// TwinCAT 3 PLC project PLC1
// ProgramVersion: 3.1.4026.16
// CompilerDefines: VISU_USEPROPERTYINFO
// libraries:
//   SH_Light, * (StroemHansen)
//   Tc2_EnOcean, * (Beckhoff Automation GmbH)
//   Tc2_Standard, * (Beckhoff Automation GmbH)
//   Tc2_System, * (Beckhoff Automation GmbH)
//   Tc2_Utilities, * (Beckhoff Automation GmbH)
//   Tc3_DALI, * (Beckhoff Automation GmbH)
//   Tc3_System_DK, * (Beckhoff - DK)
//   VisuDialogs, * (System)
// project tree:
//   DUTs/DALI/ E_DALIExtendedFadeTime.TcTLEO (not stored), ST_DALI102Parameters.TcDUT (not stored), ST_DALI103Parameters.TcDUT (not stored), ST_DALIMemoryBank.TcDUT (not stored), ST_DALI_GrpAssignment.TcDUT (not stored), ST_GroupSort.TcDUT (not stored)
//   DUTs/EnOcean/ ST_ReadSAB05.TcDUT (not stored), ST_WriteSAB05.TcDUT (not stored)
//   / FastTask.TcTTO (not stored), GlobalTextList.TcGTLO (not stored), PlcTask.TcTTO (not stored), Visualization Manager.TcVMO (not stored)
//   GVLs/ GVL_AHDataModbus.TcGVL (not stored), GVL_EnOcean.TcGVL, GVL_Skalering.TcGVL (not stored)
//   POUs/01_System/01_System/GVLs/ GVL_EtherCAT.TcGVL (not stored)
//   POUs/01_System/01_System/ P_SystemDK.TcPOU (not stored)
//   POUs/AHModbusComm/ P_AHModbusComm.TcPOU
//   POUs/Alle_Rum/Gange/Gang_1_147/ P_Gang_1_147.TcPOU (not stored), Visualization_4_330_2_1.TcVIS (not stored) (excluded from build)
//   POUs/Alle_Rum/Gange/Gang_5_441/ P_Gang_5_441.TcPOU (not stored), Visualization_4_330_1_1_1_1_2_2.TcVIS (not stored) (excluded from build)
//   POUs/Alle_Rum/Gange/Gang_7_401/ P_Gang_7_401.TcPOU, Visualization_4_330_1.TcVIS (excluded from build)
//   POUs/Alle_Rum/Gange/Gang_6_210/ P_Gang_6_210.TcPOU, Visualization_4_308_1_2_1.TcVIS (not stored) (excluded from build)
//   POUs/Alle_Rum/Gange/Gang_4_413/ P_Gang_4_413.TcPOU, Visualization_4_330.TcVIS (not stored) (excluded from build)
//   POUs/Alle_Rum/Gange/Gang_1_148/ P_Gang_1_148.TcPOU (not stored), Visualization_4_330_2.TcVIS (not stored) (excluded from build)
//   POUs/Alle_Rum/Gange/Gang_4_434A/ P_Gang_4_434A.TcPOU, Visualization_4_330_1_1_1_1_2.TcVIS (not stored) (excluded from build)
//   POUs/Alle_Rum/Gange/Gang_5_441B/ P_Gang_5_441B.TcPOU, Visualization_5_338_1_2.TcVIS (not stored) (excluded from build)
//   POUs/Alle_Rum/Gange/Gang_Atrium/ P_Gang_Atrium.TcPOU (not stored), Visualization_5_338_2.TcVIS (not stored) (excluded from build)
//   POUs/Alle_Rum/Gange/Gang_5_238/ P_Gang_5_238.TcPOU (not stored), Visualization_5_338_1.TcVIS (not stored) (excluded from build)
//   POUs/Alle_Rum/Rum_Med_DALI_Pir/1_Rum_5_125_Og_5_127_Foldedoer/ P_Foldedoer_5_125.TcPOU (not stored), P_Rum_5_127.TcPOU (not stored), P_Rum_5_125.TcPOU (not stored), Visualization_5_352_1_1_1_1_1_1.TcVIS (not stored) (excluded from build)
//   POUs/Alle_Rum/Rum_Med_DALI_Pir/Rum_4_105/ P_Rum_4_105.TcPOU, Visualization_4_330_1_1_2_1.TcVIS (not stored) (excluded from build)
//   POUs/Alle_Rum/Rum_Med_DALI_Pir/Rum_4_109D/ P_Rum_4_109D.TcPOU, Visualization_4_330_1_1_1_1_2_1_1_1_2_1_1.TcVIS (not stored) (excluded from build)
//   POUs/Alle_Rum/Rum_Med_DALI_Pir/Rum_4_111A/ P_Rum_4_111A.TcPOU, Visualization_4_330_1_1_1_1_2_1_1_1_2_1_1_1.TcVIS (excluded from build)
//   POUs/Alle_Rum/Rum_Med_DALI_Pir/1Rum_5_448A/ P_Rum_5_448A.TcPOU (not stored), Visualization_4_330_1_1_1_1_2_1_1_1_3.TcVIS (not stored) (excluded from build)
//   POUs/Alle_Rum/Rum_Med_DALI_Pir/1Rum_5_444/ P_Rum_5_444.TcPOU (not stored), Visualization_4_308_1_2_1_1.TcVIS (excluded from build)
//   POUs/Alle_Rum/Rum_Med_DALI_Pir/Rum_4_107A/ P_Rum_4_107A.TcPOU, Visualization_4_330_1_1_1_1_2_1_1_1_1.TcVIS (excluded from build)
//   POUs/Alle_Rum/Rum_Med_DALI_Pir/1Rum_5_260B/ P_Rum_5_260B.TcPOU, Visualization_4_330_1_1_1_1_2_1_1.TcVIS (excluded from build)
//   POUs/Alle_Rum/Rum_Med_DALI_Pir/1Rum_1_428/ P_Rum_1_428.TcPOU, Visualization_5_338_1_1_1_1_2_1_1_1.TcVIS (excluded from build)
//   POUs/Alle_Rum/Rum_Med_DALI_Pir/Rum_4_109A/ P_Rum_4_109A.TcPOU, Visualization_4_330_1_1_1_1_2_1_1_1_2_1.TcVIS (not stored) (excluded from build)
//   POUs/Alle_Rum/Rum_Med_DALI_Pir/1Rum_4_426/ P_Rum_4_426.TcPOU (not stored), Visualization_4_330_1_1_1_1_2_1_1_1.TcVIS (not stored) (excluded from build)
//   POUs/Alle_Rum/Rum_Med_DALI_Pir/1Rum_5_456/ P_Rum_5_456.TcPOU, Visualization_4_330_1_1_1_1_2_1_1_1_3_1_1_1_1_1.TcVIS (not stored) (excluded from build)
//   POUs/Alle_Rum/Rum_Med_DALI_Pir/1Rum_5_450/ P_Rum_5_450.TcPOU (not stored), Visualization_4_330_1_1_1_1_2_1_1_1_3_1.TcVIS (not stored) (excluded from build)
//   POUs/Alle_Rum/Rum_Med_DALI_Pir/1Rum_5_448B/ P_Rum_5_448B.TcPOU, Visualization_4_330_1_1_1_1_2_1.TcVIS (not stored) (excluded from build)
//   POUs/Alle_Rum/Rum_Med_DALI_Pir/1Rum_5_452/ P_Rum_5_452.TcPOU (not stored), Visualization_4_330_1_1_1_1_2_1_1_1_3_1_1.TcVIS (not stored) (excluded from build)
//   POUs/Alle_Rum/Rum_Med_DALI_Pir/1Rum_5_454/ P_Rum_5_454.TcPOU (not stored), Visualization_4_330_1_1_1_1_2_1_1_1_3_1_1_1.TcVIS (not stored) (excluded from build)
//   POUs/Alle_Rum/Rum_Med_DALI_Pir/1Rum_5_450B/ P_Rum_5_450B.TcPOU (not stored), Visualization_4_330_1_1_1_1_2_1_1_1_3_1_1_1_1.TcVIS (not stored) (excluded from build)
//   POUs/Alle_Rum/Rum_Med_DALI_Pir/1Rum_5_411C/ P_Rum_5_411C.TcPOU (not stored), Visualization_4_330_1_1_1_1_2_1_1_1_3_1_1_1_1_1_1.TcVIS (excluded from build)
//   POUs/Alle_Rum/Rum_Med_DALI_Pir/1Rum_6_205/ P_Rum_6_205.TcPOU (not stored), Visualization_5_338_1_1_2_1_1_1_1_1_1_1_1_1_1_1_1_2_2_1_1.TcVIS (not stored) (excluded from build)
//   POUs/Alle_Rum/Rum_Med_DALI_Pir/1Rum_5_441A/ P_Rum_5_441A.TcPOU (not stored), Visualization_5_338_1_1_2_1_1_1_1_1_1_1_1_1_1_1_1_2_2_2.TcVIS (not stored) (excluded from build)
//   POUs/Alle_Rum/Rum_Med_DALI_Pir/1Rum_5_263/ P_Rum_5_263.TcPOU (not stored), Visualization_5_338_1_1_2_1_1_1_1_1_1_1_1_1_1_1_1_2_2_1.TcVIS (excluded from build)
//   POUs/Alle_Rum/Rum_Med_DALI_Pir/1Rum_3_155/ P_Rum_3_155.TcPOU (not stored), Visualization_5_352_1_1_1_1_1_2_1.TcVIS (not stored) (excluded from build)
//   POUs/Alle_Rum/Rum_Med_DALI_Pir/1Rum_6_214B/ P_Rum_6_214B.TcPOU (not stored), Visualization_4_330_1_1_1_1_2_1_1_1_2.TcVIS (excluded from build)
//   POUs/Alle_Rum/Trapper/ P_Trappe_T4.TcPOU
//   POUs/DALI/DALI_Setup/ DALI_Commissioning.TcPOU (not stored)
//   POUs/DALI/DALI_Setup/FBs/ FB_Part102Addressing.TcPOU (not stored), FB_Part102Commands.TcPOU (not stored), FB_Part102Groups.TcPOU (not stored), FB_Part102MemoryPages.TcPOU (not stored), FB_Part102Parameters.TcPOU (not stored), FB_Part102Scenes.TcPOU (not stored), FB_Part102SetFading.TcPOU (not stored), FB_Part103Addressing.TcPOU (not stored), FB_Part103MemoryPages.TcPOU (not stored), FB_Part103Identify.TcPOU (not stored), FB_Part103Parameters.TcPOU (not stored), FB_Part202Emergency.TcPOU (not stored), FB_Part205Incandescent.TcPOU (not stored), FB_Part207LED.TcPOU (not stored), FB_Part208Switching.TcPOU (not stored), FB_Part300GenericDevice.TcPOU (not stored), FB_Part301PushButton.TcPOU (not stored), FB_Part302AbsoluteInputDevice.TcPOU (not stored), FB_Part303OccupancySensor.TcPOU (not stored), FB_Part304LightSensor.TcPOU (not stored), GearType.TcPOU (not stored)
//   POUs/DALI/DALI_Setup/GVLs/ GVL_Internal.TcGVL (not stored)
//   POUs/DALI/DALI_Setup/VISUs/TextLists/ CommandOnTerminalEvent.TcTLO (not stored), DimmingCurve.TcTLO, EventPriority.TcTLO (not stored), EventScheme.TcTLO (not stored), ExtendedFadeTime.TcTLO (not stored), FadeRate.TcTLO (not stored), FadeTime.TcTLO (not stored), FastFadeTime.TcTLO (not stored), TextList_Dialogs.TcTLO (not stored)
//   POUs/DALI/DALI_Setup/VISUs/ Visu_DALICommissioning.TcVIS (not stored)
//   POUs/DALI/DALI_Setup/VISUs/Visu_DALICommissioning/ Visu_KL6821Configuration.TcVIS (not stored) (excluded from build), Visu_Part102Addressing.TcVIS (not stored), Visu_Part102Commands.TcVIS (not stored), Visu_Part102Groups.TcVIS (not stored), Visu_Part102MemoryBank.TcVIS (not stored), Visu_Part102Parameters.TcVIS (not stored), Visu_Part102Scenes.TcVIS (not stored), Visu_Part102SetFading.TcVIS (not stored), Visu_Part103Addressing.TcVIS (not stored), Visu_Part103Identify.TcVIS (not stored), Visu_Part103MemoryBank.TcVIS (not stored), Visu_Part103Parameters.TcVIS (not stored), Visu_Part202.TcVIS (not stored), Visu_Part202Commands.TcVIS (not stored), Visu_Part202Parameters.TcVIS (not stored), Visu_Part202Status.TcVIS (not stored), Visu_Part205.TcVIS (not stored), Visu_Part205Parameters.TcVIS (not stored), Visu_Part205Status.TcVIS (not stored), Visu_Part207.TcVIS (not stored), Visu_Part207Parameters.TcVIS (not stored), Visu_Part207Status.TcVIS (not stored), Visu_Part208Switching.TcVIS (not stored), Visu_Part300GenericDevice.TcVIS (not stored), Visu_Part301PushButton.TcVIS (not stored), Visu_Part302AbsoluteInputDevice.TcVIS (not stored), Visu_Part303OccupancySensor.TcVIS (not stored), Visu_Part304LightSensor.TcVIS (not stored), Visu_Welcome.TcVIS (not stored)
//   POUs/DALI/PRGs/Background/ P_DALI_Background.TcPOU (not stored)
//   POUs/DALI/PRGs/Diag/ P_DALI_DIAG.TcPOU (not stored)
//   POUs/DALI/PRGs/EnergyData/ P_DALI_Energy_Firmware_Test.TcPOU (not stored) (excluded from build), P_DALI_Energy_Line.TcPOU (not stored)
//   POUs/EnOcean/ P_EnOcean.TcPOU
//   POUs/ MAIN.TcPOU
// real-time tasks:
//   TASK PlcTask: cycle T#40ms, priority 21, ADS port 350
//   TASK FastTask: cycle T#4ms, priority 20, ADS port 351
// I/O:
//   DEVICE Device 1 (Beckhoff CCAT)
//   DEVICE Device 3 (CX-BK)
//     Box 1 (CX-BK)
// variable links:
//   PLC1/PLC1 Instance <-> Device 3 (CX-BK)/Box 1 (CX-BK)
//     FastTask Inputs/P_DALI_Background.arrKL6821InData[1] @bit 16 <-> Term 5 (KL6821)/Channel 1/Data In 0
//     FastTask Inputs/P_DALI_Background.arrKL6821InData[1] @bit 24 <-> Term 5 (KL6821)/Channel 1/Data In 1
//     FastTask Inputs/P_DALI_Background.arrKL6821InData[1] @bit 32 <-> Term 5 (KL6821)/Channel 1/Data In 2
//     FastTask Inputs/P_DALI_Background.arrKL6821InData[1] @bit 40 <-> Term 5 (KL6821)/Channel 1/Data In 3
//     FastTask Inputs/P_DALI_Background.arrKL6821InData[2] @bit 16 <-> Term 6 (KL6821)/Channel 1/Data In 0
//     FastTask Inputs/P_DALI_Background.arrKL6821InData[2] @bit 24 <-> Term 6 (KL6821)/Channel 1/Data In 1
//     FastTask Inputs/P_DALI_Background.arrKL6821InData[2] @bit 32 <-> Term 6 (KL6821)/Channel 1/Data In 2
//     FastTask Inputs/P_DALI_Background.arrKL6821InData[2] @bit 40 <-> Term 6 (KL6821)/Channel 1/Data In 3
//     FastTask Inputs/P_DALI_Background.arrKL6821InData[1] <-> Term 5 (KL6821)/Channel 1/State
//     FastTask Inputs/P_DALI_Background.arrKL6821InData[2] <-> Term 6 (KL6821)/Channel 1/State
//     FastTask Inputs/P_EnOcean.stKL6581_in @bit 8 <-> Term 3 (KL6581)/Channel 1/Input CNODE
//     FastTask Inputs/P_EnOcean.stKL6581_in @bit {24..48 step 8} <-> Term 3 (KL6581)/Channel 1/Input DB{0..3}  (4 links)
//     FastTask Inputs/P_EnOcean.stKL6581_in @bit {56..80 step 8} <-> Term 3 (KL6581)/Channel 1/Input ID{0..3}  (4 links)
//     FastTask Inputs/P_EnOcean.stKL6581_in @bit 16 <-> Term 3 (KL6581)/Channel 1/Input ORG
//     FastTask Inputs/P_EnOcean.stKL6581_in @bit 88 <-> Term 3 (KL6581)/Channel 1/Input STATUS
//     FastTask Inputs/P_EnOcean.stKL6581_in <-> Term 3 (KL6581)/Channel 1/Status
//     FastTask Outputs/P_DALI_Background.arrKL6821OutData[1] <-> Term 5 (KL6821)/Channel 1/Ctrl
//     FastTask Outputs/P_DALI_Background.arrKL6821OutData[2] <-> Term 6 (KL6821)/Channel 1/Ctrl
//     FastTask Outputs/P_DALI_Background.arrKL6821OutData[1] @bit 16 <-> Term 5 (KL6821)/Channel 1/Data Out 0
//     FastTask Outputs/P_DALI_Background.arrKL6821OutData[1] @bit 24 <-> Term 5 (KL6821)/Channel 1/Data Out 1
//     FastTask Outputs/P_DALI_Background.arrKL6821OutData[1] @bit 32 <-> Term 5 (KL6821)/Channel 1/Data Out 2
//     FastTask Outputs/P_DALI_Background.arrKL6821OutData[1] @bit 40 <-> Term 5 (KL6821)/Channel 1/Data Out 3
//     FastTask Outputs/P_DALI_Background.arrKL6821OutData[2] @bit 16 <-> Term 6 (KL6821)/Channel 1/Data Out 0
//     FastTask Outputs/P_DALI_Background.arrKL6821OutData[2] @bit 24 <-> Term 6 (KL6821)/Channel 1/Data Out 1
//     FastTask Outputs/P_DALI_Background.arrKL6821OutData[2] @bit 32 <-> Term 6 (KL6821)/Channel 1/Data Out 2
//     FastTask Outputs/P_DALI_Background.arrKL6821OutData[2] @bit 40 <-> Term 6 (KL6821)/Channel 1/Data Out 3
//     FastTask Outputs/P_EnOcean.stKL6581_out <-> Term 3 (KL6581)/Channel 1/Control
//     FastTask Outputs/P_EnOcean.stKL6581_out @bit 8 <-> Term 3 (KL6581)/Channel 1/Output CNODE
//     FastTask Outputs/P_EnOcean.stKL6581_out @bit {24..48 step 8} <-> Term 3 (KL6581)/Channel 1/Output DB{0..3}  (4 links)
//     FastTask Outputs/P_EnOcean.stKL6581_out @bit {56..80 step 8} <-> Term 3 (KL6581)/Channel 1/Output ID{0..3}  (4 links)
//     FastTask Outputs/P_EnOcean.stKL6581_out @bit 16 <-> Term 3 (KL6581)/Channel 1/Output ORG
//     FastTask Outputs/P_EnOcean.stKL6581_out @bit 88 <-> Term 3 (KL6581)/Channel 1/Output STATUS
//     PlcTask Inputs/MAIN.nCX8200_State <-> Inputs/State
//     PlcTask Inputs/P_Trappe_T4.bDigitalPir <-> Term 4 (KL1408)/Channel 1/Input
//     PlcTask Outputs/P_Trappe_T4.bTrappelysNC <-> Term 2 (KL2012)/Channel 1/Output

// ---- GVLs/GVL_EnOcean.TcGVL
{attribute 'qualified_only'}
VAR_GLOBAL
	
//Atrium
	strEnOceanSwitch_AtriumNiveau_PladeB				: Tc2_EnOcean.STR_EnOceanSwitch;
	strEnOceanSwitch_AtriumNiveau_Service				: Tc2_EnOcean.STR_EnOceanSwitch;


//Gange
//	strEnOceanSwitch_Gang_3_364				: Tc2_EnOcean.STR_EnOceanSwitch;

	//
 
     strEnOceanSwitch_Rum_4_105                      	: Tc2_EnOcean.STR_EnOceanSwitch;


END_VAR

// ---- POUs/AHModbusComm/P_AHModbusComm.TcPOU
PROGRAM P_AHModbusComm
VAR
	arrfbReadAHPirData	: ARRAY[1..GVL_AHDataModbus.byNumberOfAH_Neighbors] OF SH_Light.FB_ReadAHPirData;
	arrReadAHPirData		: ARRAY[1..GVL_AHDataModbus.byNumberOfAH_Neighbors] OF BOOL;
	
	arrfbTriggerPulses			: ARRAY[1..GVL_AHDataModbus.byNumberOfAH_Neighbors] OF SH_Light.FB_ClockPulse;
	arrGeneratePulses			: ARRAY[1..GVL_AHDataModbus.byNumberOfAH_Neighbors] OF BOOL := [GVL_AHDataModbus.byNumberOfAH_Neighbors(TRUE)];
	tTimeInterval					: TIME := T#1S;
	tPulseTime					: TIME := T#1S;
	
	byLineId						: BYTE;
	byAHId						: BYTE;
		fbWritePirDelayTime		: R_TRIG;
	bRunOverrideOnce		: BOOL := FALSE;
	bEnableDelayTimeOverride : BOOL := FALSE;
	uiPirOffDelayTimeAllRooms : UINT := 30;
	
END_VAR

VAR CONSTANT
	arrnMBAddr					: ARRAY[1..GVL_AHDataModbus.byNumberOfAH_Neighbors] OF WORD := [GVL_AHDataModbus.byNumberOfAH_Neighbors(12588)]; //modbus-adresser (%MB600=>12588 default)
	arrstNeighborIPAddr		: ARRAY[1..GVL_AHDataModbus.byNumberOfAH_Neighbors] OF SH_Light.ST_NeighborIP := [
																						(sPLCName := 'AH1-1', sIP := '172.24.195.161', IsNeighbor := FALSE), 
																				     	(sPLCName := 'AH1-2', sIP := '172.24.195.162', IsNeighbor := FALSE), 
																						(sPLCName := 'AH1-3', sIP := '172.24.195.163', IsNeighbor := FALSE),
																						(sPLCName := 'AH2-1', sIP := '172.24.195.164', IsNeighbor := FALSE),
																					    (sPLCName := 'AH2-2', sIP := '172.24.195.165', IsNeighbor := FALSE),
																						(sPLCName := 'AH2-3', sIP := '172.24.195.166', IsNeighbor := FALSE),
																				        (sPLCName := 'AH2-4', sIP := '172.24.195.167', IsNeighbor := FALSE),
																						(sPLCName := 'AH2-5', sIP := '172.24.195.168', IsNeighbor := FALSE),
																						(sPLCName := 'AH3-2', sIP := '172.24.195.169', IsNeighbor := FALSE),
																						(sPLCName := 'AH3-3', sIP := '172.24.195.170', IsNeighbor := FALSE),
																			         	(sPLCName := 'AH3-4', sIP := '172.24.195.171', IsNeighbor := FALSE),
																						(sPLCName := 'AH3-5', sIP := '172.24.195.172', IsNeighbor := FALSE),
																						(sPLCName := 'AH4-1', sIP := '172.24.195.173', IsNeighbor := FALSE),
																						(sPLCName := 'AH4-2', sIP := '172.24.195.174', IsNeighbor := FALSE),
																						(sPLCName := 'AH4-3', sIP := '172.24.195.175', IsNeighbor := FALSE),
																			            (sPLCName := 'AH4-4', sIP := '172.24.195.176', IsNeighbor := FALSE),
																						(sPLCName := 'AH4-5', sIP := '172.24.195.177', IsNeighbor := FALSE),
																						(sPLCName := 'AH5-1', sIP := '172.24.195.178', IsNeighbor := FALSE),
																					    (sPLCName := 'AH5-2', sIP := '172.24.195.179', IsNeighbor := FALSE), 
																						(sPLCName := 'AH5-3', sIP := '172.24.195.180', IsNeighbor := FALSE),
																						(sPLCName := 'AH5-4', sIP := '172.24.195.181', IsNeighbor := FALSE),
																						(sPLCName := 'AH5-5', sIP := '172.24.195.182', IsNeighbor := FALSE),
																						(sPLCName := 'AH6-1', sIP := '172.24.195.183', IsNeighbor := FALSE),
																				        (sPLCName := 'AH6-2', sIP := '172.24.195.184', IsNeighbor := FALSE),//Local must be false
																				(sPLCName := 'AH6-3', sIP := '172.24.195.185', IsNeighbor := FALSE)];
																					//	(sPLCName := 'AH3-1', sIP := '172.24.195.186', IsNeighbor := TRUE) //when ready
END_VAR

A_AHNeighborRoomsPirIn();
A_AHNeighborRoomsPirOut();
A_DALILineShrtAddrErr();
A_DelayTimeAllRooms();

ACTION A_AHNeighborRoomsPirIn:
FOR byAHId := 1 TO GVL_AHDataModbus.byNumberOfAH_Neighbors DO
	IF arrstNeighborIPAddr[byAHId].IsNeighbor THEN
		//Generate Pulses
		arrfbTriggerPulses[byAHId](bGenerateClockPulses:= arrGeneratePulses[byAHId], tTimeInterval:= tTimeInterval, tPulseTime:= tPulseTime);
		arrReadAHPirData[byAHId]:= arrfbTriggerPulses[byAHId].bPulse;
		//Read data
		arrfbReadAHPirData[byAHId](	bReadAHPirData				:=	arrReadAHPirData[byAHId],
														sIPAddr							:=	arrstNeighborIPAddr[byAHId].sIP,
														nMBAddr							:=	arrnMBAddr[byAHId],
														nMBDataBuffer				:=	GVL_AHDataModbus.arrAH_NeighborRoomsPir_In[byAHId],
														arrAH_NeighborRoomsPir	=>GVL_AHDataModbus.arrAH_NeighborRoomsPir[byAHId]);
	END_IF
END_FOR
END_ACTION

ACTION A_AHNeighborRoomsPirOut:
//GVL_AHDataModbus.nAH_NeighborRoomsPir_Out.0 := P_Gang_4_413.bPirActive_MB;
//GVL_AHDataModbus.nAH_NeighborRoomsPir_Out.1 := P_Gang_7_401.bPirActive_MB;
//GVL_AHDataModbus.nAH_NeighborRoomsPir_Out.2 := P_Gang_5_441.bPirActive_MB;
//GVL_AHDataModbus.nAH_NeighborRoomsPir_Out.3 := P_Rum_4_424.bPirActive_MB;
//GVL_AHDataModbus.nAH_NeighborRoomsPir_Out.4 := P_Rum_4_426.bPirActive_MB;
//GVL_AHDataModbus.nAH_NeighborRoomsPir_Out.5 := 
//GVL_AHDataModbus.nAH_NeighborRoomsPir_Out.6 :=
//GVL_AHDataModbus.nAH_NeighborRoomsPir_Out.7 := 
//GVL_AHDataModbus.nAH_NeighborRoomsPir_Out.8 :=
//GVL_AHDataModbus.nAH_NeighborRoomsPir_Out.9 := 
//GVL_AHDataModbus.nAH_NeighborRoomsPir_Out.10 :=
//GVL_AHDataModbus.nAH_NeighborRoomsPir_Out.11 := 
//GVL_AHDataModbus.nAH_NeighborRoomsPir_Out.12 := 
//GVL_AHDataModbus.nAH_NeighborRoomsPir_Out.13 := 
//GVL_AHDataModbus.nAH_NeighborRoomsPir_Out.14 := 
//GVL_AHDataModbus.nAH_NeighborRoomsPir_Out.15 :=
END_ACTION

ACTION A_DALILineShrtAddrErr:
FOR  byLineId := 1 TO SH_Light.DALI_Param.MAX_DALIV2_LINES DO
	GVL_AHDataModbus.arrDALILineShrtAddrErr[byLineId] :=  TO_UINT(SH_Light.GVL_DALI_LatestError.arrLineShrtAddr[byLineId]);
END_FOR
END_ACTION

ACTION A_DelayTimeAllRooms:

fbWritePirDelayTime(CLK := GVL_AHDataModbus.uiPirOffDelayTimeAllRooms_MB<>uiPirOffDelayTimeAllRooms);

IF fbWritePirDelayTime.Q THEN
	bRunOverrideOnce := TRUE;
	bEnableDelayTimeOverride := TRUE;
	
//Indsæt kode
P_Rum_4_105.fbWritePirDelayTIme(bEnableOverride := bEnableDelayTimeOverride, nOverRideValue := GVL_AHDataModbus.uiPirOffDelayTimeAllRooms_MB, nValIn1 := GVL_AHDataModbus.uiPirOffDelayTimeAllRooms_MB, nValIn2 := uiPirOffDelayTimeAllRooms);
P_Rum_4_107A.fbWritePirDelayTIme(bEnableOverride := bEnableDelayTimeOverride, nOverRideValue := GVL_AHDataModbus.uiPirOffDelayTimeAllRooms_MB, nValIn1 := GVL_AHDataModbus.uiPirOffDelayTimeAllRooms_MB, nValIn2 := uiPirOffDelayTimeAllRooms);
P_Rum_4_109A.fbWritePirDelayTIme(bEnableOverride := bEnableDelayTimeOverride, nOverRideValue := GVL_AHDataModbus.uiPirOffDelayTimeAllRooms_MB, nValIn1 := GVL_AHDataModbus.uiPirOffDelayTimeAllRooms_MB, nValIn2 := uiPirOffDelayTimeAllRooms);
P_Rum_4_109D.fbWritePirDelayTIme(bEnableOverride := bEnableDelayTimeOverride, nOverRideValue := GVL_AHDataModbus.uiPirOffDelayTimeAllRooms_MB, nValIn1 := GVL_AHDataModbus.uiPirOffDelayTimeAllRooms_MB, nValIn2 := uiPirOffDelayTimeAllRooms);
P_Rum_4_111A.fbWritePirDelayTIme(bEnableOverride := bEnableDelayTimeOverride, nOverRideValue := GVL_AHDataModbus.uiPirOffDelayTimeAllRooms_MB, nValIn1 := GVL_AHDataModbus.uiPirOffDelayTimeAllRooms_MB, nValIn2 := uiPirOffDelayTimeAllRooms);



ELSE
	IF bRunOverrideOnce THEN
		bEnableDelayTimeOverride := FALSE;
		
		//Indsæt kode
P_Rum_4_105.fbWritePirDelayTIme(bEnableOverride := bEnableDelayTimeOverride, nOverRideValue := GVL_AHDataModbus.uiPirOffDelayTimeAllRooms_MB, nValIn1 := GVL_AHDataModbus.uiPirOffDelayTimeAllRooms_MB, nValIn2 := uiPirOffDelayTimeAllRooms);
P_Rum_4_107A.fbWritePirDelayTIme(bEnableOverride := bEnableDelayTimeOverride, nOverRideValue := GVL_AHDataModbus.uiPirOffDelayTimeAllRooms_MB, nValIn1 := GVL_AHDataModbus.uiPirOffDelayTimeAllRooms_MB, nValIn2 := uiPirOffDelayTimeAllRooms);
P_Rum_4_109A.fbWritePirDelayTIme(bEnableOverride := bEnableDelayTimeOverride, nOverRideValue := GVL_AHDataModbus.uiPirOffDelayTimeAllRooms_MB, nValIn1 := GVL_AHDataModbus.uiPirOffDelayTimeAllRooms_MB, nValIn2 := uiPirOffDelayTimeAllRooms);
P_Rum_4_109D.fbWritePirDelayTIme(bEnableOverride := bEnableDelayTimeOverride, nOverRideValue := GVL_AHDataModbus.uiPirOffDelayTimeAllRooms_MB, nValIn1 := GVL_AHDataModbus.uiPirOffDelayTimeAllRooms_MB, nValIn2 := uiPirOffDelayTimeAllRooms);
P_Rum_4_111A.fbWritePirDelayTIme(bEnableOverride := bEnableDelayTimeOverride, nOverRideValue := GVL_AHDataModbus.uiPirOffDelayTimeAllRooms_MB, nValIn1 := GVL_AHDataModbus.uiPirOffDelayTimeAllRooms_MB, nValIn2 := uiPirOffDelayTimeAllRooms);

		bRunOverrideOnce := FALSE;
		
		
	END_IF
END_IF
END_ACTION

END_PROGRAM

// ---- POUs/Alle_Rum/Rum_Med_DALI_Pir/Rum_4_105/P_Rum_4_105.TcPOU
PROGRAM P_Rum_4_105
VAR

	fbLys		: FB_Light_Type_A;
	

	stDaliSetup	: SH_Light.ST_DALI_RoomSetup := (	
														byShrtAdr_Prim := 1, 
														byGrpAdr_Prim := 1, 
														eMod_Prim := E_DALIAddressType.Group, 
														//byShrtAdr_Sec := 1, 
														//byGrpAdr_Sec := 1, 
														//eMod_Sec := E_DALIAddressType.Short, 
														//byShrtAdr_Supl := 1, 
														DALI_LINE_NUM_PRIM := DALI_LINE_NUM_LIGHT,
														DALI_LINE_NUM_SEC := 0, //0 = ingen zonestyring/vinduerække
														DALI_LINE_NUM_SUPL := DALI_LINE_NUM_PENDANTS);
														
	stLiveData					: SH_Light.ST_LiveData;
	bRunTuning					: BOOL;
	
	bTopButtonZone1				: BOOL;
	bTopButtonZone1_Visu		: BOOL;
	bBottomButtonZone1			: BOOL;
	bBottomButtonZone1_Visu	: BOOL;
	bButtonZone2				: BOOL;
	fLuxOn							: REAL;
	fLuxDim						: REAL;
	tPIRDim						: TIME;
	tPIROff						: TIME;
	fOffsetSec					: REAL := 20;
	bOccupiedRoom			: BOOL;;


// Sensor Settings
	//fbSensor						: SH_Light.FB_NIKO_P46xx_1Pcs;
	fbSensor						: SH_Light.FB_NIKO_P46xx_3Pcs;
	//bySensorAddr				: BYTE := 8;
	arrSensorAddr				: ARRAY[1..3] OF BYTE := [1,2,3];
	bInitialize						: BOOL := TRUE;
	stDaliSensorSetup			: ST_DALI_NIKOP46SetupData := (
																nSensitivityPIRSegmentA := arrSensitivityOccupancy[1],
																nSensitivityPIRSegmentB := arrSensitivityOccupancy[2],
																nSensitivityPIRSegmentC := arrSensitivityOccupancy[3]);
	//bInitErr							: BOOL;
	//bInitDone						: BOOL;
	arrInitErr						: ARRAY [1..3] OF BOOL;
	arrInitDone					: ARRAY [1..3] OF BOOL;
	arrSensorScales				: ARRAY [1..10] OF SH_Light.ST_DALI_SensorScaleMode := [
																						(fMeassureMaxSensor := rMeassure_Zone5, fReadMaxSensor := rRead_Zone5),	
																						(fMeassureMaxSensor := rMeassure_Zone5, fReadMaxSensor := rRead_Zone5),	
																						(fMeassureMaxSensor := rMeassure_Zone5, fReadMaxSensor := rRead_Zone5),																																										
																						7(())];
	bCancelHoldTimerOccupancy	: BOOL;
(*	eEventPriorityOccupancy		: E_DALIEventPriority := E_DALIEVENTPRIORITY.Middle;
	nHoldTimerOccupancy			: WORD := 5; // Value in s. 	
	nReportTimerOccupancy		: BYTE := 120; // Value in s, Preset manufacturer value
	nDeadtimeTimerOccupancy		: WORD := 100; // Value in ms, Predefined Value of DALI Standard
	bCancelHoldTimerOccupancy	: BOOL;
	nSensitivityOccupancy		: BYTE:= 3; //setting Sensivity (0..4) 0 (Off), 1 (Min), 2(Low), 3(High) and 4 (Max)

	bEnableLuxEvent				: BOOL;
	eEventPriorityBrightness	: E_DALIEventPriority := E_DALIEVENTPRIORITY.Middle;
	nDeadtimeTimerBrightness	: WORD := 1500; // Value in ms, Predefined Value of DALI Standard
	nHysteresisBrightness		: BYTE := 2; // Value in %
	nHysteresisMinBrightness	: BYTE := 10; // Absolute Value, depending on the manufacturer specific resolution
	nReportTimerBrightness		: BYTE := 120; // Value in s, Preset manufacturer value
*)

	//stDaliSetup: SH_Light.ST_DALI_RoomSetup
	//stRoomDataModbus			: SH_Light.ST_RoomDataModbus := ( bPirActive := bPirActive
	

	//ModbusComm setup
	
	fbWriteSPLuxLevel			: SH_Light.FB_TwoVal_SelectOne_RTrigChange;
	fbWritePirDelayTIme		: SH_Light.FB_TwoVal_SelectOne_RTrigChange;
	stRoomDataPLC				: SH_Light.ST_RoomDataPLC	:=	(
																	uiPirOffDelayTime	:= 30,
																	uiSpLuxLevel			:= 500,
																	uiPirDimDelayTime	:= 15,
																	uiSpDimLuxLevel		:= 200);
																	
	fbBallastOnHours				: SH_Light.FB_CountOnHours;
	bEnableHourCount			: BOOL := TRUE;
	
	//Non-persistent modbus data
	bPirActive_MB					AT %MX0.0	: BOOL;				//bPirLys i gammel kode
	uiActLuxLevel_MB			AT %MB4	: UINT;				//intHMIAktueltLux i gammel kode
	uiActLightLevelPct_MB	AT %MB10		: UINT;				//intDALI_Gruppe1_Lysniveau i gammel kode
	
	//For Conversion
	uiPirOffMinutes						: UINT;
	udTimeScaling						: UDINT := 60000;
	uiLuxOn								: UINT;
	
	//max values checks
	uiMaxLuxLevel						: UINT := 1023;
	uiMaxPirOffMinutes				: UINT := 180;

	
END_VAR

VAR CONSTANT
    Sensor_DALI_LINE_NUM				: BYTE := 1;
	DALI_LINE_NUM_LIGHT				: BYTE := 1;
    DALI_LINE_NUM_PENDANTS	: BYTE := 0; //0=ingen pendler
	arrSensitivityOccupancy						: ARRAY[1..3] OF BYTE := [4,4,4]; //setting Sensivity (0..4) 0 (Off), 1 (Min), 2(Low), 3(High) and 4 (Max)
END_VAR
VAR PERSISTENT
	stPirSensorData: SH_Light.ST_DALI_Sensor;
	stTuneData: SH_Light.ST_TuneData_EX;

	uiPirOffDelayTime_MB		AT %MB2		: UINT;				//ntHMI_Pir_SetValue i gammel kode
	uiSPLuxLevel_MB			AT %MB6	: UINT;				//intHMI_Lux_SetValue i gammel kode
	uiBallastOnHours_MB		AT %MB14		: UINT;				//dintHMILysbraendtimer1 i gammel kode
	byOnHoursOverflowCount							: BYTE;   
END_VAR

A_Buttons();
A_LightCtrl();
A_Sensor();
A_ModbusComm();

ACTION A_Buttons:
bTopButtonZone1		:= GVL_EnOcean.strEnOceanSwitch_Rum_4_105.bT1_ON OR  bTopButtonZone1_Visu;
bBottomButtonZone1	:= GVL_EnOcean.strEnOceanSwitch_Rum_4_105.bT1_OFF OR  bBottomButtonZone1_Visu;
END_ACTION

ACTION A_LightCtrl:
fbLys(
	nZoneID:= 1, 
	bButtonZone1:= bTopButtonZone1,
	bBottomButtonZone1 := bBottomButtonZone1, 
	//bButtonZone2:= bButtonZone2,
	fLuxOn:= fLuxOn, 
	fLuxDim:= fLuxDim, 
	tPIRDim:= tPIRDim, 
	tPIROff:= tPIROff, 
	fOffsetSec:= fOffsetSec, 
	bReInit:= , 
	stDaliSetup:= stDaliSetup, 
	ipCommunication_Prim:= P_DALI_Background.arrfbKL6821Communication[DALI_LINE_NUM_LIGHT], 
	//ipCommunication_Sec:= P_DALI_Background.arrfbKL6821Communication[DALI_LINE_NUM_LIGHT], 
	//ipCommunication_Supl:= P_DALI_Background.arrfbKL6821Communication[DALI_LINE_NUM_PENDANTS], 
	fMinOutputPowerLevelRoom:= 15, 
	fMaxOutputPowerLevelRoom:= 100, 
	nCycleTimeInMS:= SH_Light.DALI_Param.nPlcTaskCycleTimeInMS*nDimCmdCycleTimeFactor , 
	bRunTuning:= bRunTuning, 
	bOccupiedRoom=> bOccupiedRoom, 
	bError_Prim=> , 
	nError_Prim=> , 
	stTuneData:=stTuneData , 
	stPirSensorData:= stPirSensorData, 
	stLiveData:= stLiveData);
END_ACTION

ACTION A_ModbusComm:
//Manage data for modbus communication

//Manage data for read-only in PLC
stRoomDataPLC.bPirActive			:= stPirSensorData.bPrc;
stRoomDataPLC.uiActLuxLevel			:= TO_UINT(TRUNC(stPirSensorData.fBrightness));
stRoomDataPLC.uiActLightLevelPct	:= TO_UINT(TRUNC(fbLys.fbBallast.fActlLgtLvl_Prim));
		//stRoomDataPLC.uiActLightLevelPct	:= TO_UINT(TRUNC(fbLys.fbBallast.fActlLgtLvl_Prim)); //if only one group light control
stRoomDataPLC.uiBallastOnHours		:= uiBallastOnHours_MB; //The calculation for BallastOnHours is stored directly to the MB register below


//Assign data for read-only to MB registers
bPirActive_MB			:= stRoomDataPLC.bPirActive;
uiActLuxLevel_MB		:= stRoomDataPLC.uiActLuxLevel;
uiActLightLevelPct_MB	:= stRoomDataPLC.uiActLightLevelPct;

	//calculate BallastOnHours
	fbBallastOnHours(
		bEnableHourCount	:= bEnableHourCount,
		bPauseCount			:= fbLys.fbLightCtrl.bOffZone1,
		uiOnHours			:= uiBallastOnHours_MB,			//OnHours is updated here
		byOverflowCount		:= byOnHoursOverflowCount);


//Manage data for read/write for both PLC and MB registers
fbWriteSPLuxLevel(	nMaxValOut	:= uiMaxLuxLevel,
					nValIn1		:= uiSPLuxLevel_MB,		//nValIn1 takes priotity in case of download or restart
					nValIn2		:= stRoomDataPLC.uiSpLuxLevel,
					nValOut		=> uiLuxOn
				);


fbWritePirDelayTIme(	nMaxValOut	:= uiMaxPirOffMinutes,
						nValIn1		:= uiPirOffDelayTime_MB,		//nValIn1 takes priotity in case of download or restart
						nValIn2		:= stRoomDataPLC.uiPirOffDelayTime,
						nValOut		=> uiPirOffMinutes
					);
					

//Convert read/write modbus data to appropriate datatypes in PLC
fLuxOn	:= TO_REAL(uiLuxOn);			
tPIROff	:= TO_TIME(uiPirOffMinutes*udTimeScaling); //Time conversion defaults to ms

fLuxDim	:= TO_REAL(stRoomDataPLC.uiSpDimLuxLevel);			
tPIRDim	:= TO_TIME(stRoomDataPLC.uiPirDimDelayTime*udTimeScaling); //Time conversion defaults to ms
END_ACTION

ACTION A_Sensor:

fbSensor.ipCommunication := P_DALI_Background.arrfbKL6821Communication[Sensor_DALI_LINE_NUM];

//only 1 sensor
(*fbSensor(
	byShrtAdr:= bySensorAddr,
	bInitialize:= bInitialize, 
	DALI_LINE_NUM:= Sensor_DALI_LINE_NUM, 
 	//bCancelHoldTimerOccupancy:= bCancelHoldTimerOccupancy, 
	stSensorSetup := stDaliSensorSetup,
	bInitErr=> bInitErr, 
	bInitDone=> bInitDone,
	stPirSensorData:= stPirSensorData, 
	arrSensorScales:= arrSensorScales);
*)

//several sensors	
fbSensor(
	arrShrtAdr:= arrSensorAddr,
	bInitialize:= bInitialize, 
	DALI_LINE_NUM:= Sensor_DALI_LINE_NUM, 
 	//bCancelHoldTimerOccupancy:= bCancelHoldTimerOccupancy, 
	stSensorSetup := stDaliSensorSetup,
	arrInitErr=> arrInitErr, 
	arrInitDone=> arrInitDone,
	stPirSensorData:= stPirSensorData, 
	arrSensorScales:= arrSensorScales);
END_ACTION

END_PROGRAM

// ---- POUs/Alle_Rum/Rum_Med_DALI_Pir/Rum_4_107A/P_Rum_4_107A.TcPOU
PROGRAM P_Rum_4_107A
VAR

	fbLys		: FB_Light_Type_A;
	
	stDaliSetup	: SH_Light.ST_DALI_RoomSetup := (
														byShrtAdr_Prim := 16, 
														byGrpAdr_Prim := 2, 
														eMod_Prim := E_DALIAddressType.Group, 
														//byShrtAdr_Sec := 1, 
														//byGrpAdr_Sec := 1, 
														//eMod_Sec := E_DALIAddressType.Short, 
														//byShrtAdr_Supl := 1,
														//byGrpAdr_Supl := 1,
														//eMod_Prim := E_DALIAddressType.Short 
														DALI_LINE_NUM_PRIM := DALI_LINE_NUM_LIGHT, 
														DALI_LINE_NUM_SEC := 0, //0 = ingen zonestyring/vinduerække
														DALI_LINE_NUM_SUPL := DALI_LINE_NUM_PENDANTS);
														
	stLiveData				: SH_Light.ST_LiveData;
	bRunTuning					: BOOL;
	
	bTopButtonZone1				: BOOL;
	bTopButtonZone1_Visu		: BOOL;
	bBottomButtonZone1			: BOOL;
	bBottomButtonZone1_Visu	    : BOOL;
	bButtonZone2				: BOOL;
	bNeighborRoomsPir		    : BOOL;
	fLuxOn				     	: REAL;
	fLuxDim						: REAL;
	tPIRDim						: TIME;
	tPIROff						: TIME;
	fOffsetSec					: REAL := 20;
	bOccupiedRoom			    : BOOL;


// Sensor Settings
	fbSensor					: SH_Light.FB_NIKO_P46xx_1Pcs;
	//fbSensor					: SH_Light.FB_NIKO_P46xx_3Pcs;
	bySensorAddr				: BYTE := 4;
	//arrSensorAddr				: ARRAY[1..3] OF BYTE := [7,8,9];
	bInitialize					: BOOL := TRUE;
	stDaliSensorSetup			: ST_DALI_NIKOP46SetupData := (
																nSensitivityPIRSegmentA := arrSensitivityOccupancy[1],
																nSensitivityPIRSegmentB := arrSensitivityOccupancy[2],
																nSensitivityPIRSegmentC := arrSensitivityOccupancy[3]);
	bInitErr					: BOOL;
	bInitDone					: BOOL;
	//arrInitErr				: ARRAY [1..3] OF BOOL;
	//arrInitDone				: ARRAY [1..3] OF BOOL;
	arrSensorScales				: ARRAY [1..10] OF SH_Light.ST_DALI_SensorScaleMode := [
																						(fMeassureMaxSensor := rMeassure_Zone10, fReadMaxSensor := rRead_Zone10),																																											
																						9(())];
	bCancelHoldTimerOccupancy	: BOOL;
(*	eEventPriorityOccupancy		: E_DALIEventPriority := E_DALIEVENTPRIORITY.Middle;
	nHoldTimerOccupancy			: WORD := 5; // Value in s. 	
	nReportTimerOccupancy		: BYTE := 120; // Value in s, Preset manufacturer value
	nDeadtimeTimerOccupancy		: WORD := 100; // Value in ms, Predefined Value of DALI Standard
	bCancelHoldTimerOccupancy	: BOOL;
	nSensitivityOccupancy		: BYTE:= 3; //setting Sensivity (0..4) 0 (Off), 1 (Min), 2(Low), 3(High) and 4 (Max)

	bEnableLuxEvent				: BOOL;
	eEventPriorityBrightness	: E_DALIEventPriority := E_DALIEVENTPRIORITY.Middle;
	nDeadtimeTimerBrightness	: WORD := 1500; // Value in ms, Predefined Value of DALI Standard
	nHysteresisBrightness		: BYTE := 2; // Value in %
	nHysteresisMinBrightness	: BYTE := 10; // Absolute Value, depending on the manufacturer specific resolution
	nReportTimerBrightness		: BYTE := 120; // Value in s, Preset manufacturer value
*)

	//stDaliSetup: SH_Light.ST_DALI_RoomSetup
	//stRoomDataModbus			: SH_Light.ST_RoomDataModbus := ( bPirActive := bPirActive
	

	//ModbusComm setup
	
	fbWriteSPLuxLevel			: SH_Light.FB_TwoVal_SelectOne_RTrigChange;
	fbWritePirDelayTIme		: SH_Light.FB_TwoVal_SelectOne_RTrigChange;
	stRoomDataPLC				: SH_Light.ST_RoomDataPLC	:=	(
																	uiPirOffDelayTime	:= 30,
																	uiSpLuxLevel		:= 500,
																	uiPirDimDelayTime	:= 15,
																	uiSpDimLuxLevel		:= 200);
																	
	fbBallastOnHours				: SH_Light.FB_CountOnHours;
	bEnableHourCount			: BOOL := TRUE;
	
	//Non-persistent modbus data
	bPirActive_MB					AT %MX550.0	: BOOL;				//bPirLys i gammel kode
	uiActLuxLevel_MB			    AT %MB552	: UINT;				//intHMIAktueltLux i gammel kode
	uiActLightLevelPct_MB	        AT %MB554	: UINT;				//intDALI_Gruppe1_Lysniveau i gammel kode
	
	//For Conversion
	uiPirOffMinutes						: UINT;
	udTimeScaling						: UDINT := 60000;
	uiLuxOn								: UINT;
	
	//max values checks
	uiMaxLuxLevel						: UINT := 1023;
	uiMaxPirOffMinutes				    : UINT := 180;

	
END_VAR

VAR CONSTANT
    Sensor_DALI_LINE_NUM				: BYTE := 1;
	DALI_LINE_NUM_LIGHT			     	: BYTE := 1;
	DALI_LINE_NUM_PENDANTS	            : BYTE := 0; //0=ingen pendler	
	arrSensitivityOccupancy				: ARRAY[1..3] OF BYTE := [4,4,4]; //sensitivitet for sensor
END_VAR
VAR PERSISTENT
	stPirSensorData: SH_Light.ST_DALI_Sensor;
	stTuneData: SH_Light.ST_TuneData_EX;

	uiPirOffDelayTime_MB	AT %MB556	: UINT;				//ntHMI_Pir_SetValue i gammel kode
	uiSPLuxLevel_MB			AT %MB558	: UINT;				//intHMI_Lux_SetValue i gammel kode
	uiBallastOnHours_MB		AT %MB560	: UINT;				//dintHMILysbraendtimer1 i gammel kode
	byOnHoursOverflowCount				: BYTE;   
END_VAR

A_Buttons();
A_LightCtrl();
A_Sensor();
A_ModbusComm();

ACTION A_Buttons:
//bTopButtonZone1		:= GVL_EnOcean.strEnOceanSwitch_Rum_4_107A.bT2_ON OR bTopButtonZone1_Visu;
//bBottomButtonZone1	:= GVL_EnOcean.strEnOceanSwitch_Rum_4_107A.bT2_OFF OR bBottomButtonZone1_Visu;
END_ACTION

ACTION A_LightCtrl:

fbLys(
	nZoneID:= 1, 
	bButtonZone1:= bTopButtonZone1,
	bBottomButtonZone1 := bBottomButtonZone1, 
	//bButtonZone2:= bButtonZone2,
	fLuxOn:= fLuxOn, 
	fLuxDim:= fLuxDim, 
	tPIRDim:= tPIRDim, 
	tPIROff:= tPIROff, 
	fOffsetSec:= fOffsetSec, 
	bReInit:= , 
	stDaliSetup:= stDaliSetup, 
	ipCommunication_Prim:= P_DALI_Background.arrfbKL6821Communication[DALI_LINE_NUM_LIGHT], 
	//ipCommunication_Sec:= P_DALI_Background.arrfbKL6821Communication[DALI_LINE_NUM_LIGHT], 
	//ipCommunication_Supl:= P_DALI_Background.arrfbKL6821Communication[DALI_LINE_NUM_PENDANTS], 
	fMinOutputPowerLevelRoom:= 15, 
	fMaxOutputPowerLevelRoom:= 100, 
	nCycleTimeInMS:= SH_Light.DALI_Param.nPlcTaskCycleTimeInMS*nDimCmdCycleTimeFactor , 
	bRunTuning:= bRunTuning, 
	bOccupiedRoom=> bOccupiedRoom, 
	bError_Prim=> , 
	nError_Prim=> , 
	stTuneData:=stTuneData , 
	stPirSensorData:= stPirSensorData, 
	stLiveData:= stLiveData);
END_ACTION

ACTION A_ModbusComm:
//Manage data for modbus communication

//Manage data for read-only in PLC
stRoomDataPLC.bPirActive			:= stPirSensorData.bPrc;
stRoomDataPLC.uiActLuxLevel			:= TO_UINT(TRUNC(stPirSensorData.fBrightness));
stRoomDataPLC.uiActLightLevelPct	:= TO_UINT(TRUNC(fbLys.fbBallast.fActlLgtLvl_Prim));
		//stRoomDataPLC.uiActLightLevelPct	:= TO_UINT(TRUNC(fbLys.fbBallast.fActlLgtLvl_Prim)); //if only one group light control
stRoomDataPLC.uiBallastOnHours		:= uiBallastOnHours_MB; //The calculation for BallastOnHours is stored directly to the MB register below


//Assign data for read-only to MB registers
bPirActive_MB			:= stRoomDataPLC.bPirActive;
uiActLuxLevel_MB		:= stRoomDataPLC.uiActLuxLevel;
uiActLightLevelPct_MB	:= stRoomDataPLC.uiActLightLevelPct;

	//calculate BallastOnHours
	fbBallastOnHours(
		bEnableHourCount	:= bEnableHourCount,
		bPauseCount			:= fbLys.fbLightCtrl.bOffZone1,
		uiOnHours			:= uiBallastOnHours_MB,			//OnHours is updated here
		byOverflowCount		:= byOnHoursOverflowCount);


//Manage data for read/write for both PLC and MB registers
fbWriteSPLuxLevel(	nMaxValOut	:= uiMaxLuxLevel,
					nValIn1		:= uiSPLuxLevel_MB,		//nValIn1 takes priotity in case of download or restart
					nValIn2		:= stRoomDataPLC.uiSpLuxLevel,
					nValOut		=> uiLuxOn
				);


fbWritePirDelayTIme(	nMaxValOut	:= uiMaxPirOffMinutes,
						nValIn1		:= uiPirOffDelayTime_MB,		//nValIn1 takes priotity in case of download or restart
						nValIn2		:= stRoomDataPLC.uiPirOffDelayTime,
						nValOut		=> uiPirOffMinutes
					);
					

//Convert read/write modbus data to appropriate datatypes in PLC
fLuxOn	:= TO_REAL(uiLuxOn);			
tPIROff	:= TO_TIME(uiPirOffMinutes*udTimeScaling); //Time conversion defaults to ms

fLuxDim	:= TO_REAL(stRoomDataPLC.uiSpDimLuxLevel);			
tPIRDim	:= TO_TIME(stRoomDataPLC.uiPirDimDelayTime*udTimeScaling); //Time conversion defaults to ms
END_ACTION

ACTION A_Sensor:

fbSensor.ipCommunication := P_DALI_Background.arrfbKL6821Communication[Sensor_DALI_LINE_NUM];

//only 1 sensor
fbSensor(
	byShrtAdr:= bySensorAddr,
	bInitialize:= bInitialize, 
	DALI_LINE_NUM:= Sensor_DALI_LINE_NUM, 
 	//bCancelHoldTimerOccupancy:= bCancelHoldTimerOccupancy, 
	stSensorSetup := stDaliSensorSetup,
	bInitErr=> bInitErr, 
	bInitDone=> bInitDone,
	stPirSensorData:= stPirSensorData, 
	arrSensorScales:= arrSensorScales);


(*//several sensors	
fbSensor(
	arrShrtAdr:= arrSensorAddr,
	bInitialize:= bInitialize, 
	DALI_LINE_NUM:= Sensor_DALI_LINE_NUM, 
 	//bCancelHoldTimerOccupancy:= bCancelHoldTimerOccupancy, 
	stSensorSetup := stDaliSensorSetup,
	arrInitErr=> arrInitErr, 
	arrInitDone=> arrInitDone,
	stPirSensorData:= stPirSensorData, 
	arrSensorScales:= arrSensorScales);
	*)
END_ACTION

END_PROGRAM

// ---- POUs/Alle_Rum/Rum_Med_DALI_Pir/Rum_4_109A/P_Rum_4_109A.TcPOU
PROGRAM P_Rum_4_109A
VAR

	fbLys		: FB_Light_Type_A;
	
	stDaliSetup	: SH_Light.ST_DALI_RoomSetup := (
														byShrtAdr_Prim := 3, 
														byGrpAdr_Prim := 2, 
														eMod_Prim := E_DALIAddressType.Group, 
														//byShrtAdr_Sec := 1, 
														//byGrpAdr_Sec := 1, 
														//eMod_Sec := E_DALIAddressType.Short, 
														//eMod_Supl := E_DALIADDRESSTYPE.Short,
														//byShrtAdr_Supl := 22,
														DALI_LINE_NUM_PRIM := DALI_LINE_NUM_LIGHT, 
														DALI_LINE_NUM_SEC := 0, //0 = ingen zonestyring/vinduerække
														DALI_LINE_NUM_SUPL := DALI_LINE_NUM_PENDANTS);
														
	stLiveData				: SH_Light.ST_LiveData;
	bRunTuning					: BOOL;
	
	bTopButtonZone1				: BOOL;
	bTopButtonZone1_Visu		: BOOL;
	bBottomButtonZone1			: BOOL;
	bBottomButtonZone1_Visu	    : BOOL;
	bButtonZone2				: BOOL;
	bNeighborRoomsPir		    : BOOL;
	fLuxOn				     	: REAL;
	fLuxDim						: REAL;
	tPIRDim						: TIME;
	tPIROff						: TIME;
	fOffsetSec					: REAL := 20;
	bOccupiedRoom			    : BOOL;


// Sensor Settings
	fbSensor					: SH_Light.FB_NIKO_P46xx_1Pcs;
	//fbSensor					: SH_Light.FB_NIKO_P46xx_3Pcs;
	bySensorAddr				: BYTE := 2;
	//arrSensorAddr				: ARRAY[1..3] OF BYTE := [7,8,9];
	bInitialize					: BOOL := TRUE;
	stDaliSensorSetup			: ST_DALI_NIKOP46SetupData := (
																nSensitivityPIRSegmentA := arrSensitivityOccupancy[1],
																nSensitivityPIRSegmentB := arrSensitivityOccupancy[2],
																nSensitivityPIRSegmentC := arrSensitivityOccupancy[3]);
	bInitErr					: BOOL;
	bInitDone					: BOOL;
	//arrInitErr				: ARRAY [1..3] OF BOOL;
	//arrInitDone				: ARRAY [1..3] OF BOOL;
	arrSensorScales				: ARRAY [1..10] OF SH_Light.ST_DALI_SensorScaleMode := [
																						(fMeassureMaxSensor := rMeassure_Zone10, fReadMaxSensor := rRead_Zone10),																																									
																						9(())];
	bCancelHoldTimerOccupancy	: BOOL;
(*	eEventPriorityOccupancy		: E_DALIEventPriority := E_DALIEVENTPRIORITY.Middle;
	nHoldTimerOccupancy			: WORD := 5; // Value in s. 	
	nReportTimerOccupancy		: BYTE := 120; // Value in s, Preset manufacturer value
	nDeadtimeTimerOccupancy		: WORD := 100; // Value in ms, Predefined Value of DALI Standard
	bCancelHoldTimerOccupancy	: BOOL;
	nSensitivityOccupancy		: BYTE:= 3; //setting Sensivity (0..4) 0 (Off), 1 (Min), 2(Low), 3(High) and 4 (Max)

	bEnableLuxEvent				: BOOL;
	eEventPriorityBrightness	: E_DALIEventPriority := E_DALIEVENTPRIORITY.Middle;
	nDeadtimeTimerBrightness	: WORD := 1500; // Value in ms, Predefined Value of DALI Standard
	nHysteresisBrightness		: BYTE := 2; // Value in %
	nHysteresisMinBrightness	: BYTE := 10; // Absolute Value, depending on the manufacturer specific resolution
	nReportTimerBrightness		: BYTE := 120; // Value in s, Preset manufacturer value
*)

	//stDaliSetup: SH_Light.ST_DALI_RoomSetup
	//stRoomDataModbus			: SH_Light.ST_RoomDataModbus := ( bPirActive := bPirActive
	

	//ModbusComm setup
	
	fbWriteSPLuxLevel			: SH_Light.FB_TwoVal_SelectOne_RTrigChange;
	fbWritePirDelayTIme		: SH_Light.FB_TwoVal_SelectOne_RTrigChange;
	stRoomDataPLC				: SH_Light.ST_RoomDataPLC	:=	(
																	uiPirOffDelayTime	:= 30,
																	uiSpLuxLevel		:= 500,
																	uiPirDimDelayTime	:= 15,
																	uiSpDimLuxLevel		:= 200);
																	
	fbBallastOnHours				: SH_Light.FB_CountOnHours;
	bEnableHourCount			: BOOL := TRUE;
	
	//Non-persistent modbus data
	bPirActive_MB					AT %MX30.0	: BOOL;				//bPirLys i gammel kode
	uiActLuxLevel_MB			    AT %MB540	: UINT;				//intHMIAktueltLux i gammel kode
	uiActLightLevelPct_MB	        AT %MB34	: UINT;				//intDALI_Gruppe1_Lysniveau i gammel kode
	
	//For Conversion
	uiPirOffMinutes						: UINT;
	udTimeScaling						: UDINT := 60000;
	uiLuxOn								: UINT;
	
	//max values checks
	uiMaxLuxLevel						: UINT := 1023;
	uiMaxPirOffMinutes				    : UINT := 180;

	
END_VAR

VAR CONSTANT
    Sensor_DALI_LINE_NUM				: BYTE := 2;
	DALI_LINE_NUM_LIGHT			     	: BYTE := 2;
	DALI_LINE_NUM_PENDANTS	            : BYTE := 0; //0=ingen pendler	
	arrSensitivityOccupancy				: ARRAY[1..3] OF BYTE := [4,4,4]; //sensitivitet for sensor
END_VAR
VAR PERSISTENT
	stPirSensorData: SH_Light.ST_DALI_Sensor;
	stTuneData: SH_Light.ST_TuneData_EX;

	uiPirOffDelayTime_MB	AT %MB32	: UINT;				//ntHMI_Pir_SetValue i gammel kode
	uiSPLuxLevel_MB			AT %MB542	: UINT;				//intHMI_Lux_SetValue i gammel kode
	uiBallastOnHours_MB		AT %MB36	: UINT;				//dintHMILysbraendtimer1 i gammel kode
	byOnHoursOverflowCount				: BYTE;   
END_VAR

A_Buttons();
A_LightCtrl();
A_Sensor();
A_ModbusComm();

ACTION A_Buttons:
bTopButtonZone1		:= bTopButtonZone1_Visu;
bBottomButtonZone1	:= bBottomButtonZone1_Visu;
END_ACTION

ACTION A_LightCtrl:

fbLys(
	nZoneID:= 1, 
	bButtonZone1:= bTopButtonZone1,
	bBottomButtonZone1 := bBottomButtonZone1, 
	bButtonZone2:= bButtonZone2,
	fLuxOn:= fLuxOn, 
	fLuxDim:= fLuxDim, 
	tPIRDim:= tPIRDim, 
	tPIROff:= tPIROff, 
	fOffsetSec:= fOffsetSec, 
	bReInit:= , 
	stDaliSetup:= stDaliSetup, 
	ipCommunication_Prim:= P_DALI_Background.arrfbKL6821Communication[DALI_LINE_NUM_LIGHT], 
	//ipCommunication_Sec:= P_DALI_Background.arrfbKL6821Communication[DALI_LINE_NUM_LIGHT], 
	//ipCommunication_Supl:= P_DALI_Background.arrfbKL6821Communication[DALI_LINE_NUM_PENDANTS], 
	fMinOutputPowerLevelRoom:= 15, 
	fMaxOutputPowerLevelRoom:= 100, 
	nCycleTimeInMS:= SH_Light.DALI_Param.nPlcTaskCycleTimeInMS*nDimCmdCycleTimeFactor , 
	bRunTuning:= bRunTuning, 
	bOccupiedRoom=> bOccupiedRoom, 
	bError_Prim=> , 
	nError_Prim=> , 
	stTuneData:=stTuneData , 
	stPirSensorData:= stPirSensorData, 
	stLiveData:= stLiveData);
END_ACTION

ACTION A_ModbusComm:
//Manage data for modbus communication

//Manage data for read-only in PLC
stRoomDataPLC.bPirActive			:= stPirSensorData.bPrc;
stRoomDataPLC.uiActLuxLevel			:= TO_UINT(TRUNC(stPirSensorData.fBrightness));
stRoomDataPLC.uiActLightLevelPct	:= TO_UINT(TRUNC(fbLys.fbBallast.fActlLgtLvl_Prim));
		//stRoomDataPLC.uiActLightLevelPct	:= TO_UINT(TRUNC(fbLys.fbBallast.fActlLgtLvl_Prim)); //if only one group light control
stRoomDataPLC.uiBallastOnHours		:= uiBallastOnHours_MB; //The calculation for BallastOnHours is stored directly to the MB register below


//Assign data for read-only to MB registers
bPirActive_MB			:= stRoomDataPLC.bPirActive;
uiActLuxLevel_MB		:= stRoomDataPLC.uiActLuxLevel;
uiActLightLevelPct_MB	:= stRoomDataPLC.uiActLightLevelPct;

	//calculate BallastOnHours
	fbBallastOnHours(
		bEnableHourCount	:= bEnableHourCount,
		bPauseCount			:= fbLys.fbLightCtrl.bOffZone1,
		uiOnHours			:= uiBallastOnHours_MB,			//OnHours is updated here
		byOverflowCount		:= byOnHoursOverflowCount);


//Manage data for read/write for both PLC and MB registers
fbWriteSPLuxLevel(	nMaxValOut	:= uiMaxLuxLevel,
					nValIn1		:= uiSPLuxLevel_MB,		//nValIn1 takes priotity in case of download or restart
					nValIn2		:= stRoomDataPLC.uiSpLuxLevel,
					nValOut		=> uiLuxOn
				);


fbWritePirDelayTIme(	nMaxValOut	:= uiMaxPirOffMinutes,
						nValIn1		:= uiPirOffDelayTime_MB,		//nValIn1 takes priotity in case of download or restart
						nValIn2		:= stRoomDataPLC.uiPirOffDelayTime,
						nValOut		=> uiPirOffMinutes
					);
					

//Convert read/write modbus data to appropriate datatypes in PLC
fLuxOn	:= TO_REAL(uiLuxOn);			
tPIROff	:= TO_TIME(uiPirOffMinutes*udTimeScaling); //Time conversion defaults to ms

fLuxDim	:= TO_REAL(stRoomDataPLC.uiSpDimLuxLevel);			
tPIRDim	:= TO_TIME(stRoomDataPLC.uiPirDimDelayTime*udTimeScaling); //Time conversion defaults to ms
END_ACTION

ACTION A_Sensor:

fbSensor.ipCommunication := P_DALI_Background.arrfbKL6821Communication[Sensor_DALI_LINE_NUM];

//only 1 sensor
fbSensor(
	byShrtAdr:= bySensorAddr,
	bInitialize:= bInitialize, 
	DALI_LINE_NUM:= Sensor_DALI_LINE_NUM, 
 	//bCancelHoldTimerOccupancy:= bCancelHoldTimerOccupancy, 
	stSensorSetup := stDaliSensorSetup,
	bInitErr=> bInitErr, 
	bInitDone=> bInitDone,
	stPirSensorData:= stPirSensorData, 
	arrSensorScales:= arrSensorScales);


(*//several sensors	
fbSensor(
	arrShrtAdr:= arrSensorAddr,
	bInitialize:= bInitialize, 
	DALI_LINE_NUM:= Sensor_DALI_LINE_NUM, 
 	//bCancelHoldTimerOccupancy:= bCancelHoldTimerOccupancy, 
	stSensorSetup := stDaliSensorSetup,
	arrInitErr=> arrInitErr, 
	arrInitDone=> arrInitDone,
	stPirSensorData:= stPirSensorData, 
	arrSensorScales:= arrSensorScales);
	*)
END_ACTION

END_PROGRAM

// ---- POUs/Alle_Rum/Rum_Med_DALI_Pir/Rum_4_109D/P_Rum_4_109D.TcPOU
PROGRAM P_Rum_4_109D
VAR

	fbLys		: FB_Light_Type_A;
	
	stDaliSetup	: SH_Light.ST_DALI_RoomSetup := (
														byShrtAdr_Prim := 1, 
														byGrpAdr_Prim := 1, 
														eMod_Prim := E_DALIAddressType.Group, 
														//byShrtAdr_Sec := 1, 
														//byGrpAdr_Sec := 1, 
														//eMod_Sec := E_DALIAddressType.Short, 
														//eMod_Supl := E_DALIADDRESSTYPE.Short,
														//byShrtAdr_Supl := 22,
														DALI_LINE_NUM_PRIM := DALI_LINE_NUM_LIGHT, 
														DALI_LINE_NUM_SEC := 0, //0 = ingen zonestyring/vinduerække
														DALI_LINE_NUM_SUPL := DALI_LINE_NUM_PENDANTS);
														
	stLiveData				: SH_Light.ST_LiveData;
	bRunTuning					: BOOL;
	
	bTopButtonZone1				: BOOL;
	bTopButtonZone1_Visu		: BOOL;
	bBottomButtonZone1			: BOOL;
	bBottomButtonZone1_Visu	    : BOOL;
	bButtonZone2				: BOOL;
	bNeighborRoomsPir		    : BOOL;
	fLuxOn				     	: REAL;
	fLuxDim						: REAL;
	tPIRDim						: TIME;
	tPIROff						: TIME;
	fOffsetSec					: REAL := 20;
	bOccupiedRoom			    : BOOL;


// Sensor Settings
	fbSensor					: SH_Light.FB_NIKO_P46xx_1Pcs;
	//fbSensor					: SH_Light.FB_NIKO_P46xx_3Pcs;
	bySensorAddr				: BYTE := 1;
	//arrSensorAddr				: ARRAY[1..3] OF BYTE := [7,8,9];
	bInitialize					: BOOL := TRUE;
	stDaliSensorSetup			: ST_DALI_NIKOP46SetupData := (
																nSensitivityPIRSegmentA := arrSensitivityOccupancy[1],
																nSensitivityPIRSegmentB := arrSensitivityOccupancy[2],
																nSensitivityPIRSegmentC := arrSensitivityOccupancy[3]);
	bInitErr					: BOOL;
	bInitDone					: BOOL;
	//arrInitErr				: ARRAY [1..3] OF BOOL;
	//arrInitDone				: ARRAY [1..3] OF BOOL;
	arrSensorScales				: ARRAY [1..10] OF SH_Light.ST_DALI_SensorScaleMode := [
																						(fMeassureMaxSensor := rMeassure_Zone10, fReadMaxSensor := rRead_Zone10),																																										
																						9(())];
	bCancelHoldTimerOccupancy	: BOOL;
(*	eEventPriorityOccupancy		: E_DALIEventPriority := E_DALIEVENTPRIORITY.Middle;
	nHoldTimerOccupancy			: WORD := 5; // Value in s. 	
	nReportTimerOccupancy		: BYTE := 120; // Value in s, Preset manufacturer value
	nDeadtimeTimerOccupancy		: WORD := 100; // Value in ms, Predefined Value of DALI Standard
	bCancelHoldTimerOccupancy	: BOOL;
	nSensitivityOccupancy		: BYTE:= 3; //setting Sensivity (0..4) 0 (Off), 1 (Min), 2(Low), 3(High) and 4 (Max)

	bEnableLuxEvent				: BOOL;
	eEventPriorityBrightness	: E_DALIEventPriority := E_DALIEVENTPRIORITY.Middle;
	nDeadtimeTimerBrightness	: WORD := 1500; // Value in ms, Predefined Value of DALI Standard
	nHysteresisBrightness		: BYTE := 2; // Value in %
	nHysteresisMinBrightness	: BYTE := 10; // Absolute Value, depending on the manufacturer specific resolution
	nReportTimerBrightness		: BYTE := 120; // Value in s, Preset manufacturer value
*)

	//stDaliSetup: SH_Light.ST_DALI_RoomSetup
	//stRoomDataModbus			: SH_Light.ST_RoomDataModbus := ( bPirActive := bPirActive
	

	//ModbusComm setup
	
	fbWriteSPLuxLevel			: SH_Light.FB_TwoVal_SelectOne_RTrigChange;
	fbWritePirDelayTIme		: SH_Light.FB_TwoVal_SelectOne_RTrigChange;
	stRoomDataPLC				: SH_Light.ST_RoomDataPLC	:=	(
																	uiPirOffDelayTime	:= 30,
																	uiSpLuxLevel		:= 500,
																	uiPirDimDelayTime	:= 15,
																	uiSpDimLuxLevel		:= 200);
																	
	fbBallastOnHours				: SH_Light.FB_CountOnHours;
	bEnableHourCount			: BOOL := TRUE;
	
	//Non-persistent modbus data
	bPirActive_MB					AT %MX38.0	: BOOL;				//bPirLys i gammel kode
	uiActLuxLevel_MB			    AT %MB42	: UINT;				//intHMIAktueltLux i gammel kode
	uiActLightLevelPct_MB	        AT %MB46	: UINT;				//intDALI_Gruppe1_Lysniveau i gammel kode
	
	//For Conversion
	uiPirOffMinutes						: UINT;
	udTimeScaling						: UDINT := 60000;
	uiLuxOn								: UINT;
	
	//max values checks
	uiMaxLuxLevel						: UINT := 1023;
	uiMaxPirOffMinutes				    : UINT := 180;

	
END_VAR

VAR CONSTANT
    Sensor_DALI_LINE_NUM				: BYTE := 2;
	DALI_LINE_NUM_LIGHT			     	: BYTE := 2;
	DALI_LINE_NUM_PENDANTS	            : BYTE := 0; //0=ingen pendler	
	arrSensitivityOccupancy				: ARRAY[1..3] OF BYTE := [4,4,4]; //sensitivitet for sensor
END_VAR
VAR PERSISTENT
	stPirSensorData: SH_Light.ST_DALI_Sensor;
	stTuneData: SH_Light.ST_TuneData_EX;

	uiPirOffDelayTime_MB	AT %MB40	: UINT;				//ntHMI_Pir_SetValue i gammel kode
	uiSPLuxLevel_MB			AT %MB44	: UINT;				//intHMI_Lux_SetValue i gammel kode
	uiBallastOnHours_MB		AT %MB48	: UINT;				//dintHMILysbraendtimer1 i gammel kode
	byOnHoursOverflowCount				: BYTE;   
END_VAR

A_Buttons();
A_LightCtrl();
A_Sensor();
A_ModbusComm();

ACTION A_Buttons:
bTopButtonZone1		:= bTopButtonZone1_Visu;
bBottomButtonZone1	:= bBottomButtonZone1_Visu;
END_ACTION

ACTION A_LightCtrl:

fbLys(
	nZoneID:= 1, 
	bButtonZone1:= bTopButtonZone1,
	bBottomButtonZone1 := bBottomButtonZone1, 
	bButtonZone2:= bButtonZone2,
	fLuxOn:= fLuxOn, 
	fLuxDim:= fLuxDim, 
	tPIRDim:= tPIRDim, 
	tPIROff:= tPIROff, 
	fOffsetSec:= fOffsetSec, 
	bReInit:= , 
	stDaliSetup:= stDaliSetup, 
	ipCommunication_Prim:= P_DALI_Background.arrfbKL6821Communication[DALI_LINE_NUM_LIGHT], 
	//ipCommunication_Sec:= P_DALI_Background.arrfbKL6821Communication[DALI_LINE_NUM_LIGHT], 
	//ipCommunication_Supl:= P_DALI_Background.arrfbKL6821Communication[DALI_LINE_NUM_PENDANTS], 
	fMinOutputPowerLevelRoom:= 15, 
	fMaxOutputPowerLevelRoom:= 100, 
	nCycleTimeInMS:= SH_Light.DALI_Param.nPlcTaskCycleTimeInMS*nDimCmdCycleTimeFactor , 
	bRunTuning:= bRunTuning, 
	bOccupiedRoom=> bOccupiedRoom, 
	bError_Prim=> , 
	nError_Prim=> , 
	stTuneData:=stTuneData , 
	stPirSensorData:= stPirSensorData, 
	stLiveData:= stLiveData);
END_ACTION

ACTION A_ModbusComm:
//Manage data for modbus communication

//Manage data for read-only in PLC
stRoomDataPLC.bPirActive			:= stPirSensorData.bPrc;
stRoomDataPLC.uiActLuxLevel			:= TO_UINT(TRUNC(stPirSensorData.fBrightness));
stRoomDataPLC.uiActLightLevelPct	:= TO_UINT(TRUNC(fbLys.fbBallast.fActlLgtLvl_Prim));
		//stRoomDataPLC.uiActLightLevelPct	:= TO_UINT(TRUNC(fbLys.fbBallast.fActlLgtLvl_Prim)); //if only one group light control
stRoomDataPLC.uiBallastOnHours		:= uiBallastOnHours_MB; //The calculation for BallastOnHours is stored directly to the MB register below


//Assign data for read-only to MB registers
bPirActive_MB			:= stRoomDataPLC.bPirActive;
uiActLuxLevel_MB		:= stRoomDataPLC.uiActLuxLevel;
uiActLightLevelPct_MB	:= stRoomDataPLC.uiActLightLevelPct;

	//calculate BallastOnHours
	fbBallastOnHours(
		bEnableHourCount	:= bEnableHourCount,
		bPauseCount			:= fbLys.fbLightCtrl.bOffZone1,
		uiOnHours			:= uiBallastOnHours_MB,			//OnHours is updated here
		byOverflowCount		:= byOnHoursOverflowCount);


//Manage data for read/write for both PLC and MB registers
fbWriteSPLuxLevel(	nMaxValOut	:= uiMaxLuxLevel,
					nValIn1		:= uiSPLuxLevel_MB,		//nValIn1 takes priotity in case of download or restart
					nValIn2		:= stRoomDataPLC.uiSpLuxLevel,
					nValOut		=> uiLuxOn
				);


fbWritePirDelayTIme(	nMaxValOut	:= uiMaxPirOffMinutes,
						nValIn1		:= uiPirOffDelayTime_MB,		//nValIn1 takes priotity in case of download or restart
						nValIn2		:= stRoomDataPLC.uiPirOffDelayTime,
						nValOut		=> uiPirOffMinutes
					);
					

//Convert read/write modbus data to appropriate datatypes in PLC
fLuxOn	:= TO_REAL(uiLuxOn);			
tPIROff	:= TO_TIME(uiPirOffMinutes*udTimeScaling); //Time conversion defaults to ms

fLuxDim	:= TO_REAL(stRoomDataPLC.uiSpDimLuxLevel);			
tPIRDim	:= TO_TIME(stRoomDataPLC.uiPirDimDelayTime*udTimeScaling); //Time conversion defaults to ms
END_ACTION

ACTION A_Sensor:

fbSensor.ipCommunication := P_DALI_Background.arrfbKL6821Communication[Sensor_DALI_LINE_NUM];

//only 1 sensor
fbSensor(
	byShrtAdr:= bySensorAddr,
	bInitialize:= bInitialize, 
	DALI_LINE_NUM:= Sensor_DALI_LINE_NUM, 
 	//bCancelHoldTimerOccupancy:= bCancelHoldTimerOccupancy, 
	stSensorSetup := stDaliSensorSetup,
	bInitErr=> bInitErr, 
	bInitDone=> bInitDone,
	stPirSensorData:= stPirSensorData, 
	arrSensorScales:= arrSensorScales);


(*//several sensors	
fbSensor(
	arrShrtAdr:= arrSensorAddr,
	bInitialize:= bInitialize, 
	DALI_LINE_NUM:= Sensor_DALI_LINE_NUM, 
 	//bCancelHoldTimerOccupancy:= bCancelHoldTimerOccupancy, 
	stSensorSetup := stDaliSensorSetup,
	arrInitErr=> arrInitErr, 
	arrInitDone=> arrInitDone,
	stPirSensorData:= stPirSensorData, 
	arrSensorScales:= arrSensorScales);
	*)
END_ACTION

END_PROGRAM

// ---- POUs/Alle_Rum/Rum_Med_DALI_Pir/Rum_4_111A/P_Rum_4_111A.TcPOU
PROGRAM P_Rum_4_111A
VAR

	fbLys		: FB_Light_Type_A;
	
	stDaliSetup	: SH_Light.ST_DALI_RoomSetup := (
														byShrtAdr_Prim := 6, 
														byGrpAdr_Prim := 3, 
														eMod_Prim := E_DALIAddressType.Group, 
														//byShrtAdr_Sec := 1, 
														//byGrpAdr_Sec := 1, 
														//eMod_Sec := E_DALIAddressType.Short, 
														//eMod_Supl := E_DALIADDRESSTYPE.Short,
														//byShrtAdr_Supl := 22,
														DALI_LINE_NUM_PRIM := DALI_LINE_NUM_LIGHT, 
														DALI_LINE_NUM_SEC := 0, //0 = ingen zonestyring/vinduerække
														DALI_LINE_NUM_SUPL := DALI_LINE_NUM_PENDANTS);
														
	stLiveData				: SH_Light.ST_LiveData;
	bRunTuning					: BOOL;
	
	bTopButtonZone1				: BOOL;
	bTopButtonZone1_Visu		: BOOL;
	bBottomButtonZone1			: BOOL;
	bBottomButtonZone1_Visu	    : BOOL;
	bButtonZone2				: BOOL;
	bNeighborRoomsPir		    : BOOL;
	fLuxOn				     	: REAL;
	fLuxDim						: REAL;
	tPIRDim						: TIME;
	tPIROff						: TIME;
	fOffsetSec					: REAL := 20;
	bOccupiedRoom			    : BOOL;


// Sensor Settings
	fbSensor					: SH_Light.FB_NIKO_P46xx_1Pcs;
	//fbSensor					: SH_Light.FB_NIKO_P46xx_3Pcs;
	bySensorAddr				: BYTE := 3;
	//arrSensorAddr				: ARRAY[1..3] OF BYTE := [7,8,9];
	bInitialize					: BOOL := TRUE;
	stDaliSensorSetup			: ST_DALI_NIKOP46SetupData := (
																nSensitivityPIRSegmentA := arrSensitivityOccupancy[1],
																nSensitivityPIRSegmentB := arrSensitivityOccupancy[2],
																nSensitivityPIRSegmentC := arrSensitivityOccupancy[3]);
	bInitErr					: BOOL;
	bInitDone					: BOOL;
	//arrInitErr				: ARRAY [1..3] OF BOOL;
	//arrInitDone				: ARRAY [1..3] OF BOOL;
	arrSensorScales				: ARRAY [1..10] OF SH_Light.ST_DALI_SensorScaleMode := [
																						(fMeassureMaxSensor := rMeassure_Zone10, fReadMaxSensor := rRead_Zone10),																																									
																						9(())];
	bCancelHoldTimerOccupancy	: BOOL;
(*	eEventPriorityOccupancy		: E_DALIEventPriority := E_DALIEVENTPRIORITY.Middle;
	nHoldTimerOccupancy			: WORD := 5; // Value in s. 	
	nReportTimerOccupancy		: BYTE := 120; // Value in s, Preset manufacturer value
	nDeadtimeTimerOccupancy		: WORD := 100; // Value in ms, Predefined Value of DALI Standard
	bCancelHoldTimerOccupancy	: BOOL;
	nSensitivityOccupancy		: BYTE:= 3; //setting Sensivity (0..4) 0 (Off), 1 (Min), 2(Low), 3(High) and 4 (Max)

	bEnableLuxEvent				: BOOL;
	eEventPriorityBrightness	: E_DALIEventPriority := E_DALIEVENTPRIORITY.Middle;
	nDeadtimeTimerBrightness	: WORD := 1500; // Value in ms, Predefined Value of DALI Standard
	nHysteresisBrightness		: BYTE := 2; // Value in %
	nHysteresisMinBrightness	: BYTE := 10; // Absolute Value, depending on the manufacturer specific resolution
	nReportTimerBrightness		: BYTE := 120; // Value in s, Preset manufacturer value
*)

	//stDaliSetup: SH_Light.ST_DALI_RoomSetup
	//stRoomDataModbus			: SH_Light.ST_RoomDataModbus := ( bPirActive := bPirActive
	

	//ModbusComm setup
	
	fbWriteSPLuxLevel			: SH_Light.FB_TwoVal_SelectOne_RTrigChange;
	fbWritePirDelayTIme		: SH_Light.FB_TwoVal_SelectOne_RTrigChange;
	stRoomDataPLC				: SH_Light.ST_RoomDataPLC	:=	(
																	uiPirOffDelayTime	:= 30,
																	uiSpLuxLevel		:= 500,
																	uiPirDimDelayTime	:= 15,
																	uiSpDimLuxLevel		:= 200);
																	
	fbBallastOnHours				: SH_Light.FB_CountOnHours;
	bEnableHourCount			: BOOL := TRUE;
	
	//Non-persistent modbus data
	bPirActive_MB					AT %MX50.0	: BOOL;				//bPirLys i gammel kode
	uiActLuxLevel_MB			    AT %MB54	: UINT;				//intHMIAktueltLux i gammel kode
	uiActLightLevelPct_MB	        AT %MB58	: UINT;				//intDALI_Gruppe1_Lysniveau i gammel kode
	
	//For Conversion
	uiPirOffMinutes						: UINT;
	udTimeScaling						: UDINT := 60000;
	uiLuxOn								: UINT;
	
	//max values checks
	uiMaxLuxLevel						: UINT := 1023;
	uiMaxPirOffMinutes				    : UINT := 180;

	
END_VAR

VAR CONSTANT
    Sensor_DALI_LINE_NUM				: BYTE := 2;
	DALI_LINE_NUM_LIGHT			     	: BYTE := 2;
	DALI_LINE_NUM_PENDANTS	            : BYTE := 0; //0=ingen pendler	
	arrSensitivityOccupancy				: ARRAY[1..3] OF BYTE := [4,4,4]; //sensitivitet for sensor
END_VAR
VAR PERSISTENT
	stPirSensorData: SH_Light.ST_DALI_Sensor;
	stTuneData: SH_Light.ST_TuneData_EX;

	uiPirOffDelayTime_MB	AT %MB52	: UINT;				//ntHMI_Pir_SetValue i gammel kode
	uiSPLuxLevel_MB			AT %MB56	: UINT;				//intHMI_Lux_SetValue i gammel kode
	uiBallastOnHours_MB		AT %MB60	: UINT;				//dintHMILysbraendtimer1 i gammel kode
	byOnHoursOverflowCount				: BYTE;   
END_VAR

A_Buttons();
A_LightCtrl();
A_Sensor();
A_ModbusComm();

ACTION A_Buttons:
bTopButtonZone1		:= bTopButtonZone1_Visu;
bBottomButtonZone1	:= bBottomButtonZone1_Visu;
END_ACTION

ACTION A_LightCtrl:

fbLys(
	nZoneID:= 1, 
	bButtonZone1:= bTopButtonZone1,
	bBottomButtonZone1 := bBottomButtonZone1, 
	bButtonZone2:= bButtonZone2,
	fLuxOn:= fLuxOn, 
	fLuxDim:= fLuxDim, 
	tPIRDim:= tPIRDim, 
	tPIROff:= tPIROff, 
	fOffsetSec:= fOffsetSec, 
	bReInit:= , 
	stDaliSetup:= stDaliSetup, 
	ipCommunication_Prim:= P_DALI_Background.arrfbKL6821Communication[DALI_LINE_NUM_LIGHT], 
	//ipCommunication_Sec:= P_DALI_Background.arrfbKL6821Communication[DALI_LINE_NUM_LIGHT], 
	//ipCommunication_Supl:= P_DALI_Background.arrfbKL6821Communication[DALI_LINE_NUM_PENDANTS], 
	fMinOutputPowerLevelRoom:= 15, 
	fMaxOutputPowerLevelRoom:= 100, 
	nCycleTimeInMS:= SH_Light.DALI_Param.nPlcTaskCycleTimeInMS*nDimCmdCycleTimeFactor , 
	bRunTuning:= bRunTuning, 
	bOccupiedRoom=> bOccupiedRoom, 
	bError_Prim=> , 
	nError_Prim=> , 
	stTuneData:=stTuneData , 
	stPirSensorData:= stPirSensorData, 
	stLiveData:= stLiveData);
END_ACTION

ACTION A_ModbusComm:
//Manage data for modbus communication

//Manage data for read-only in PLC
stRoomDataPLC.bPirActive			:= stPirSensorData.bPrc;
stRoomDataPLC.uiActLuxLevel			:= TO_UINT(TRUNC(stPirSensorData.fBrightness));
stRoomDataPLC.uiActLightLevelPct	:= TO_UINT(TRUNC(fbLys.fbBallast.fActlLgtLvl_Prim));
		//stRoomDataPLC.uiActLightLevelPct	:= TO_UINT(TRUNC(fbLys.fbBallast.fActlLgtLvl_Prim)); //if only one group light control
stRoomDataPLC.uiBallastOnHours		:= uiBallastOnHours_MB; //The calculation for BallastOnHours is stored directly to the MB register below


//Assign data for read-only to MB registers
bPirActive_MB			:= stRoomDataPLC.bPirActive;
uiActLuxLevel_MB		:= stRoomDataPLC.uiActLuxLevel;
uiActLightLevelPct_MB	:= stRoomDataPLC.uiActLightLevelPct;

	//calculate BallastOnHours
	fbBallastOnHours(
		bEnableHourCount	:= bEnableHourCount,
		bPauseCount			:= fbLys.fbLightCtrl.bOffZone1,
		uiOnHours			:= uiBallastOnHours_MB,			//OnHours is updated here
		byOverflowCount		:= byOnHoursOverflowCount);


//Manage data for read/write for both PLC and MB registers
fbWriteSPLuxLevel(	nMaxValOut	:= uiMaxLuxLevel,
					nValIn1		:= uiSPLuxLevel_MB,		//nValIn1 takes priotity in case of download or restart
					nValIn2		:= stRoomDataPLC.uiSpLuxLevel,
					nValOut		=> uiLuxOn
				);


fbWritePirDelayTIme(	nMaxValOut	:= uiMaxPirOffMinutes,
						nValIn1		:= uiPirOffDelayTime_MB,		//nValIn1 takes priotity in case of download or restart
						nValIn2		:= stRoomDataPLC.uiPirOffDelayTime,
						nValOut		=> uiPirOffMinutes
					);
					

//Convert read/write modbus data to appropriate datatypes in PLC
fLuxOn	:= TO_REAL(uiLuxOn);			
tPIROff	:= TO_TIME(uiPirOffMinutes*udTimeScaling); //Time conversion defaults to ms

fLuxDim	:= TO_REAL(stRoomDataPLC.uiSpDimLuxLevel);			
tPIRDim	:= TO_TIME(stRoomDataPLC.uiPirDimDelayTime*udTimeScaling); //Time conversion defaults to ms
END_ACTION

ACTION A_Sensor:

fbSensor.ipCommunication := P_DALI_Background.arrfbKL6821Communication[Sensor_DALI_LINE_NUM];

//only 1 sensor
fbSensor(
	byShrtAdr:= bySensorAddr,
	bInitialize:= bInitialize, 
	DALI_LINE_NUM:= Sensor_DALI_LINE_NUM, 
 	//bCancelHoldTimerOccupancy:= bCancelHoldTimerOccupancy, 
	stSensorSetup := stDaliSensorSetup,
	bInitErr=> bInitErr, 
	bInitDone=> bInitDone,
	stPirSensorData:= stPirSensorData, 
	arrSensorScales:= arrSensorScales);


(*//several sensors	
fbSensor(
	arrShrtAdr:= arrSensorAddr,
	bInitialize:= bInitialize, 
	DALI_LINE_NUM:= Sensor_DALI_LINE_NUM, 
 	//bCancelHoldTimerOccupancy:= bCancelHoldTimerOccupancy, 
	stSensorSetup := stDaliSensorSetup,
	arrInitErr=> arrInitErr, 
	arrInitDone=> arrInitDone,
	stPirSensorData:= stPirSensorData, 
	arrSensorScales:= arrSensorScales);
	*)
END_ACTION

END_PROGRAM

// ---- POUs/Alle_Rum/Gange/Gang_7_401/P_Gang_7_401.TcPOU
PROGRAM P_Gang_7_401
VAR

	fbLys		: FB_Light_Type_B;
	

	stDaliSetup	: SH_Light.ST_DALI_RoomSetup := (
														byShrtAdr_Prim := 40, 
														byGrpAdr_Prim := 2, 
														eMod_Prim := E_DALIAddressType.Group, 
														//byShrtAdr_Sec := 1, 
														//byGrpAdr_Sec := 1, 
														//eMod_Sec := E_DALIAddressType.Short, 
														//byShrtAdr_Supl := 19, 
														DALI_LINE_NUM_PRIM := DALI_LINE_NUM_LIGHT,
														DALI_LINE_NUM_SEC := 0, //0 = ingen zonestyring/vinduerække
													    DALI_LINE_NUM_SUPL := DALI_LINE_NUM_PENDANTS);
														
	stLiveData				: SH_Light.ST_LiveData;
	bRunTuning					: BOOL;
	
	bTopButtonZone1				: BOOL;
	bTopButtonZone1_Visu		: BOOL;
	bBottomButtonZone1			: BOOL;
	bBottomButtonZone1_Visu	    : BOOL;
	bButtonZone2				: BOOL;
	bNeighborRoomsPir			: BOOL;
	fLuxOn						: REAL;
	fLuxDim						: REAL;
	tPIRDim						: TIME;
	tPIROff						: TIME;
	fOffsetSec					: REAL := 20;
	bOccupiedRoom				: BOOL;;


// Sensor Settings
	//fbSensor					: SH_Light.FB_NIKO_P46xx_1Pcs;
	fbSensor					: SH_Light.FB_NIKO_P46xx_4Pcs;
	//bySensorAddr				: BYTE := 1;
	arrSensorAddr				: ARRAY[1..4] OF BYTE := [3,4,5,6];
	bInitialize					: BOOL := TRUE;
	stDaliSensorSetup			: ST_DALI_NIKOP46SetupData := (
																nSensitivityPIRSegmentA := arrSensitivityOccupancy[1],
																nSensitivityPIRSegmentB := arrSensitivityOccupancy[2],
																nSensitivityPIRSegmentC := arrSensitivityOccupancy[3]);
	//bInitErr					: BOOL;
	//bInitDone					: BOOL;
	arrInitErr					: ARRAY [1..4] OF BOOL;
	arrInitDone					: ARRAY [1..4] OF BOOL;
	arrSensorScales				: ARRAY [1..10] OF SH_Light.ST_DALI_SensorScaleMode := [
																						(fMeassureMaxSensor := 1023, fReadMaxSensor := 1023),
																						(fMeassureMaxSensor := 1023, fReadMaxSensor := 1023),
																						(fMeassureMaxSensor := 1023, fReadMaxSensor := 1023),
																						(fMeassureMaxSensor := 1023, fReadMaxSensor := 1023),																																												
																						6(())];
																						
	bCancelHoldTimerOccupancy	: BOOL;
(*	eEventPriorityOccupancy		: E_DALIEventPriority := E_DALIEVENTPRIORITY.Middle;
	nHoldTimerOccupancy			: WORD := 5; // Value in s. 	
	nReportTimerOccupancy		: BYTE := 120; // Value in s, Preset manufacturer value
	nDeadtimeTimerOccupancy		: WORD := 100; // Value in ms, Predefined Value of DALI Standard
	bCancelHoldTimerOccupancy	: BOOL;
	nSensitivityOccupancy		: BYTE:= 3; //setting Sensivity (0..4) 0 (Off), 1 (Min), 2(Low), 3(High) and 4 (Max)

	bEnableLuxEvent				: BOOL;
	eEventPriorityBrightness	: E_DALIEventPriority := E_DALIEVENTPRIORITY.Middle;
	nDeadtimeTimerBrightness	: WORD := 1500; // Value in ms, Predefined Value of DALI Standard
	nHysteresisBrightness		: BYTE := 2; // Value in %
	nHysteresisMinBrightness	: BYTE := 10; // Absolute Value, depending on the manufacturer specific resolution
	nReportTimerBrightness		: BYTE := 120; // Value in s, Preset manufacturer value
*)
	

	//ModbusComm setup
	
	fbWriteSPLuxLevel				: SH_Light.FB_TwoVal_SelectOne_RTrigChange;
	fbWritePirDelayTIme			: SH_Light.FB_TwoVal_SelectOne_RTrigChange;
	stRoomDataPLC					: SH_Light.ST_RoomDataPLC	:=	(
																	uiPirOffDelayTime	:= 30,
																	uiSpLuxLevel			:= 500,
																	uiPirDimDelayTime	:= 15,
																	uiSpDimLuxLevel		:= 200);
																	
	fbBallastOnHours				: SH_Light.FB_CountOnHours;
	bEnableHourCount			: BOOL := TRUE;
	
	//Non-persistent modbus data
	bPirActive_MB				AT %MX505.0	: BOOL;				//bPirLys i gammel kode
	uiActLuxLevel_MB			AT %MB518	: UINT;				//intHMIAktueltLux i gammel kode
	uiActLightLevelPct_MB	    AT %MB522	: UINT;				//intDALI_Gruppe1_Lysniveau i gammel kode
	
	//For Conversion
	uiPirOffMinutes						: UINT;
	udTimeScaling						: UDINT := 60000;
	uiLuxOn								: UINT;
	
	//max values checks
	uiMaxLuxLevel						: UINT := 1023;
	uiMaxPirOffMinutes			    	: UINT := 180;

	
END_VAR

VAR CONSTANT
    Sensor_DALI_LINE_NUM				: BYTE := 4;
	DALI_LINE_NUM_LIGHT			    	: BYTE := 1;
	DALI_LINE_NUM_PENDANTS	            : BYTE := 0; //0=ingen pendler
	arrSensitivityOccupancy				: ARRAY[1..3] OF BYTE := [4,4,4];
END_VAR
VAR PERSISTENT
	stPirSensorData: SH_Light.ST_DALI_Sensor;
	stTuneData: SH_Light.ST_TuneData_EX;

	uiPirOffDelayTime_MB	AT %MB516	: UINT;				//ntHMI_Pir_SetValue i gammel kode
	uiSPLuxLevel_MB			AT %MB520	: UINT;				//intHMI_Lux_SetValue i gammel kode
	uiBallastOnHours_MB		AT %MB524	: UINT;				//dintHMILysbraendtimer1 i gammel kode
	byOnHoursOverflowCount				: BYTE;   
END_VAR

A_Buttons();
A_LightCtrl();
A_Sensor();
A_ModbusComm();

ACTION A_Buttons:
bTopButtonZone1		:= bTopButtonZone1_Visu;
bBottomButtonZone1	:= bBottomButtonZone1_Visu;
END_ACTION

ACTION A_LightCtrl:
bNeighborRoomsPir	:= P_Gang_4_413.stPirSensorData.bPrc              OR
                       GVL_AHDataModbus.arrAH_NeighborRoomsPir[7][1] OR
					   GVL_AHDataModbus.arrAH_NeighborRoomsPir[11][0] OR
                       GVL_AHDataModbus.arrAH_NeighborRoomsPir[11][2]  ;


fbLys(
	nZoneID:= 1, 
	bButtonZone1:= bTopButtonZone1, 
	bBottomButtonZone1 := bBottomButtonZone1,
	bButtonZone2:= bButtonZone2,
	bTopButtonOverride := (GVL_EnOcean.strEnOceanSwitch_AtriumNiveau_PladeB.bT2_ON ),
	bBottomButtonOverride := (GVL_EnOcean.strEnOceanSwitch_AtriumNiveau_PladeB.bT2_OFF ),
	bNoButtons := TRUE,
	bNeighborRoomsPir	:=	bNeighborRoomsPir,
	fLuxOn:= fLuxOn, 
	fLuxDim:= fLuxDim, 
	tPIRDim:= tPIRDim, 
	tPIROff:= tPIROff, 
	fOffsetSec:= fOffsetSec, 
	bReInit:= , 
	stDaliSetup:= stDaliSetup, 
	ipCommunication_Prim:= P_DALI_Background.arrfbKL6821Communication[DALI_LINE_NUM_LIGHT], 
	//ipCommunication_Sec:= P_DALI_Background.arrfbKL6821Communication[DALI_LINE_NUM_LIGHT], 
	//ipCommunication_Supl:= P_DALI_Background.arrfbKL6821Communication[DALI_LINE_NUM_PENDANTS], 
	fMinOutputPowerLevelRoom:= 15, 
	fMaxOutputPowerLevelRoom:= 100, 
	nCycleTimeInMS:= SH_Light.DALI_Param.nPlcTaskCycleTimeInMS*nDimCmdCycleTimeFactor , 
	bRunTuning:= bRunTuning, 
	bOccupiedRoom=> bOccupiedRoom, 
	bError_Prim=> , 
	nError_Prim=> , 
	stTuneData:=stTuneData , 
	stPirSensorData:= stPirSensorData, 
	stLiveData:= stLiveData);
END_ACTION

ACTION A_ModbusComm:
//Manage data for modbus communication

//Manage data for read-only in PLC
stRoomDataPLC.bPirActive			:= stPirSensorData.bPrc;
stRoomDataPLC.uiActLuxLevel			:= TO_UINT(TRUNC(stPirSensorData.fBrightness));
stRoomDataPLC.uiActLightLevelPct	:= TO_UINT(TRUNC(fbLys.fbBallast.fActlLgtLvl_Prim));
		//stRoomDataPLC.uiActLightLevelPct	:= TO_UINT(TRUNC(fbLys.fbBallast.fActlLgtLvl_Prim)); //if only one group light control
stRoomDataPLC.uiBallastOnHours		:= uiBallastOnHours_MB; //The calculation for BallastOnHours is stored directly to the MB register below


//Assign data for read-only to MB registers
bPirActive_MB			:= stRoomDataPLC.bPirActive;
uiActLuxLevel_MB		:= stRoomDataPLC.uiActLuxLevel;
uiActLightLevelPct_MB	:= stRoomDataPLC.uiActLightLevelPct;

	//calculate BallastOnHours
	fbBallastOnHours(
		bEnableHourCount	:= bEnableHourCount,
		bPauseCount			:= fbLys.fbLightCtrl.bOffZone1,
		uiOnHours			:= uiBallastOnHours_MB,			//OnHours is updated here
		byOverflowCount		:= byOnHoursOverflowCount);


//Manage data for read/write for both PLC and MB registers
fbWriteSPLuxLevel(	nMaxValOut	:= uiMaxLuxLevel,
					nValIn1		:= uiSPLuxLevel_MB,		//nValIn1 takes priotity in case of download or restart
					nValIn2		:= stRoomDataPLC.uiSpLuxLevel,
					nValOut		=> uiLuxOn
				);


fbWritePirDelayTIme(	nMaxValOut	:= uiMaxPirOffMinutes,
						nValIn1		:= uiPirOffDelayTime_MB,		//nValIn1 takes priotity in case of download or restart
						nValIn2		:= stRoomDataPLC.uiPirOffDelayTime,
						nValOut		=> uiPirOffMinutes
					);
					

//Convert read/write modbus data to appropriate datatypes in PLC
fLuxOn	:= TO_REAL(uiLuxOn);			
tPIROff	:= TO_TIME(uiPirOffMinutes*udTimeScaling); //Time conversion defaults to ms

fLuxDim	:= TO_REAL(stRoomDataPLC.uiSpDimLuxLevel);			
tPIRDim	:= TO_TIME(stRoomDataPLC.uiPirDimDelayTime*udTimeScaling); //Time conversion defaults to ms
END_ACTION

ACTION A_Sensor:

fbSensor.ipCommunication := P_DALI_Background.arrfbKL6821Communication[Sensor_DALI_LINE_NUM];

//only 1 sensor 
(*
fbSensor(
	byShrtAdr:= bySensorAddr,
	bInitialize:= bInitialize, 
	DALI_LINE_NUM:= Sensor_DALI_LINE_NUM, 
 	//bCancelHoldTimerOccupancy:= bCancelHoldTimerOccupancy, 
	stSensorSetup := stDaliSensorSetup,
	bInitErr=> bInitErr, 
	bInitDone=> bInitDone,
	stPirSensorData:= stPirSensorData, 
	arrSensorScales:= arrSensorScales);

*)
//several sensors	
fbSensor(
	arrShrtAdr:= arrSensorAddr,
	bInitialize:= bInitialize, 
	DALI_LINE_NUM:= Sensor_DALI_LINE_NUM, 
 	//bCancelHoldTimerOccupancy:= bCancelHoldTimerOccupancy, 
	stSensorSetup := stDaliSensorSetup,
	arrInitErr=> arrInitErr, 
	arrInitDone=> arrInitDone,
	stPirSensorData:= stPirSensorData, 
	arrSensorScales:= arrSensorScales);
END_ACTION

END_PROGRAM

// ---- POUs/Alle_Rum/Gange/Gang_4_413/P_Gang_4_413.TcPOU
PROGRAM P_Gang_4_413
VAR

	fbLys		: FB_Light_Type_B;
	

	stDaliSetup	: SH_Light.ST_DALI_RoomSetup := (
														byShrtAdr_Prim := 1, 
														byGrpAdr_Prim := 1, 
														eMod_Prim := E_DALIAddressType.Group, 
														//byShrtAdr_Sec := 1, 
														//byGrpAdr_Sec := 1, 
														//eMod_Sec := E_DALIAddressType.Short, 
														//byShrtAdr_Supl := 19, 
														DALI_LINE_NUM_PRIM := DALI_LINE_NUM_LIGHT,
														DALI_LINE_NUM_SEC := 0, //0 = ingen zonestyring/vinduerække
													    DALI_LINE_NUM_SUPL := DALI_LINE_NUM_PENDANTS);
														
	stLiveData				: SH_Light.ST_LiveData;
	bRunTuning					: BOOL;
	
	bTopButtonZone1				: BOOL;
	bTopButtonZone1_Visu		: BOOL;
	bBottomButtonZone1			: BOOL;
	bBottomButtonZone1_Visu	    : BOOL;
	bButtonZone2				: BOOL;
	bNeighborRoomsPir			: BOOL;
	fLuxOn						: REAL;
	fLuxDim						: REAL;
	tPIRDim						: TIME;
	tPIROff						: TIME;
	fOffsetSec					: REAL := 20;
	bOccupiedRoom				: BOOL;;


// Sensor Settings
	//fbSensor					: SH_Light.FB_NIKO_P46xx_1Pcs;
	fbSensor					: SH_Light.FB_NIKO_P46xx_5Pcs;
	//bySensorAddr				: BYTE := 1;
	arrSensorAddr				: ARRAY[1..5] OF BYTE := [1,2,3,4,5];
	bInitialize					: BOOL := TRUE;
	stDaliSensorSetup			: ST_DALI_NIKOP46SetupData := (
																nSensitivityPIRSegmentA := arrSensitivityOccupancy[1],
																nSensitivityPIRSegmentB := arrSensitivityOccupancy[2],
																nSensitivityPIRSegmentC := arrSensitivityOccupancy[3]);
	//bInitErr					: BOOL;
	//bInitDone					: BOOL;
	arrInitErr					: ARRAY [1..5] OF BOOL;
	arrInitDone					: ARRAY [1..5] OF BOOL;
	arrSensorScales				: ARRAY [1..10] OF SH_Light.ST_DALI_SensorScaleMode := [
																						(fMeassureMaxSensor := 1023, fReadMaxSensor := 1023),
																						(fMeassureMaxSensor := 1023, fReadMaxSensor := 1023),
																						(fMeassureMaxSensor := 1023, fReadMaxSensor := 1023),
																						(fMeassureMaxSensor := 1023, fReadMaxSensor := 1023),	
																						(fMeassureMaxSensor := 1023, fReadMaxSensor := 1023),																																												
																						5(())];
																						
	bCancelHoldTimerOccupancy	: BOOL;
(*	eEventPriorityOccupancy		: E_DALIEventPriority := E_DALIEVENTPRIORITY.Middle;
	nHoldTimerOccupancy			: WORD := 5; // Value in s. 	
	nReportTimerOccupancy		: BYTE := 120; // Value in s, Preset manufacturer value
	nDeadtimeTimerOccupancy		: WORD := 100; // Value in ms, Predefined Value of DALI Standard
	bCancelHoldTimerOccupancy	: BOOL;
	nSensitivityOccupancy		: BYTE:= 3; //setting Sensivity (0..4) 0 (Off), 1 (Min), 2(Low), 3(High) and 4 (Max)

	bEnableLuxEvent				: BOOL;
	eEventPriorityBrightness	: E_DALIEventPriority := E_DALIEVENTPRIORITY.Middle;
	nDeadtimeTimerBrightness	: WORD := 1500; // Value in ms, Predefined Value of DALI Standard
	nHysteresisBrightness		: BYTE := 2; // Value in %
	nHysteresisMinBrightness	: BYTE := 10; // Absolute Value, depending on the manufacturer specific resolution
	nReportTimerBrightness		: BYTE := 120; // Value in s, Preset manufacturer value
*)
	

	//ModbusComm setup
	
	fbWriteSPLuxLevel				: SH_Light.FB_TwoVal_SelectOne_RTrigChange;
	fbWritePirDelayTIme			: SH_Light.FB_TwoVal_SelectOne_RTrigChange;
	stRoomDataPLC					: SH_Light.ST_RoomDataPLC	:=	(
																	uiPirOffDelayTime	:= 30,
																	uiSpLuxLevel			:= 500,
																	uiPirDimDelayTime	:= 15,
																	uiSpDimLuxLevel		:= 200);
																	
	fbBallastOnHours				: SH_Light.FB_CountOnHours;
	bEnableHourCount			: BOOL := TRUE;
	
	//Non-persistent modbus data
	bPirActive_MB				AT %MX500.0	: BOOL;				//bPirLys i gammel kode
	uiActLuxLevel_MB			AT %MB508	: UINT;				//intHMIAktueltLux i gammel kode
	uiActLightLevelPct_MB	    AT %MB512	: UINT;				//intDALI_Gruppe1_Lysniveau i gammel kode
	
	//For Conversion
	uiPirOffMinutes						: UINT;
	udTimeScaling						: UDINT := 60000;
	uiLuxOn								: UINT;
	
	//max values checks
	uiMaxLuxLevel						: UINT := 1023;
	uiMaxPirOffMinutes			    	: UINT := 180;

	
END_VAR

VAR CONSTANT
    Sensor_DALI_LINE_NUM				: BYTE := 3;
	DALI_LINE_NUM_LIGHT			    	: BYTE := 1;
	DALI_LINE_NUM_PENDANTS	            : BYTE := 0; //0=ingen pendler
	arrSensitivityOccupancy				: ARRAY[1..3] OF BYTE := [4,4,4];
END_VAR
VAR PERSISTENT
	stPirSensorData: SH_Light.ST_DALI_Sensor;
	stTuneData: SH_Light.ST_TuneData_EX;

	uiPirOffDelayTime_MB	AT %MB506	: UINT;				//ntHMI_Pir_SetValue i gammel kode
	uiSPLuxLevel_MB			AT %MB510	: UINT;				//intHMI_Lux_SetValue i gammel kode
	uiBallastOnHours_MB		AT %MB514	: UINT;				//dintHMILysbraendtimer1 i gammel kode
	byOnHoursOverflowCount				: BYTE;   
END_VAR

A_Buttons();
A_LightCtrl();
A_Sensor();
A_ModbusComm();

ACTION A_Buttons:
bTopButtonZone1		:= bTopButtonZone1_Visu;
bBottomButtonZone1	:= bBottomButtonZone1_Visu;
END_ACTION

ACTION A_LightCtrl:
bNeighborRoomsPir	:= P_Gang_7_401.stPirSensorData.bPrc              OR
                       P_Gang_5_441B.stPirSensorData.bPrc             OR
					   P_Gang_4_434A.stPirSensorData.bPrc             OR
					   P_Rum_4_424.stPirSensorData.bPrc               OR
					   P_Rum_4_426.stPirSensorData.bPrc               OR
                       GVL_AHDataModbus.arrAH_NeighborRoomsPir[15][1] OR
					   GVL_AHDataModbus.arrAH_NeighborRoomsPir[7][1]
;
fbLys(
	nZoneID:= 1, 
	bButtonZone1:= bTopButtonZone1, 
	bBottomButtonZone1 := bBottomButtonZone1,
	bButtonZone2:= bButtonZone2,
	bTopButtonOverride := (GVL_EnOcean.strEnOceanSwitch_AtriumNiveau_PladeB.bT2_ON),
	bBottomButtonOverride := (GVL_EnOcean.strEnOceanSwitch_AtriumNiveau_PladeB.bT2_OFF),
	bNoButtons := TRUE,
	bNeighborRoomsPir	:=	bNeighborRoomsPir,
	fLuxOn:= fLuxOn, 
	fLuxDim:= fLuxDim, 
	tPIRDim:= tPIRDim, 
	tPIROff:= tPIROff, 
	fOffsetSec:= fOffsetSec, 
	bReInit:= , 
	stDaliSetup:= stDaliSetup, 
	ipCommunication_Prim:= P_DALI_Background.arrfbKL6821Communication[DALI_LINE_NUM_LIGHT], 
	//ipCommunication_Sec:= P_DALI_Background.arrfbKL6821Communication[DALI_LINE_NUM_LIGHT], 
	//ipCommunication_Supl:= P_DALI_Background.arrfbKL6821Communication[DALI_LINE_NUM_PENDANTS], 
	fMinOutputPowerLevelRoom:= 15, 
	fMaxOutputPowerLevelRoom:= 100, 
	nCycleTimeInMS:= SH_Light.DALI_Param.nPlcTaskCycleTimeInMS*nDimCmdCycleTimeFactor , 
	bRunTuning:= bRunTuning, 
	bOccupiedRoom=> bOccupiedRoom, 
	bError_Prim=> , 
	nError_Prim=> , 
	stTuneData:=stTuneData , 
	stPirSensorData:= stPirSensorData, 
	stLiveData:= stLiveData);
END_ACTION

ACTION A_ModbusComm:
//Manage data for modbus communication

//Manage data for read-only in PLC
stRoomDataPLC.bPirActive			:= stPirSensorData.bPrc;
stRoomDataPLC.uiActLuxLevel			:= TO_UINT(TRUNC(stPirSensorData.fBrightness));
stRoomDataPLC.uiActLightLevelPct	:= TO_UINT(TRUNC(fbLys.fbBallast.fActlLgtLvl_Prim));
		//stRoomDataPLC.uiActLightLevelPct	:= TO_UINT(TRUNC(fbLys.fbBallast.fActlLgtLvl_Prim)); //if only one group light control
stRoomDataPLC.uiBallastOnHours		:= uiBallastOnHours_MB; //The calculation for BallastOnHours is stored directly to the MB register below


//Assign data for read-only to MB registers
bPirActive_MB			:= stRoomDataPLC.bPirActive;
uiActLuxLevel_MB		:= stRoomDataPLC.uiActLuxLevel;
uiActLightLevelPct_MB	:= stRoomDataPLC.uiActLightLevelPct;

	//calculate BallastOnHours
	fbBallastOnHours(
		bEnableHourCount	:= bEnableHourCount,
		bPauseCount			:= fbLys.fbLightCtrl.bOffZone1,
		uiOnHours			:= uiBallastOnHours_MB,			//OnHours is updated here
		byOverflowCount		:= byOnHoursOverflowCount);


//Manage data for read/write for both PLC and MB registers
fbWriteSPLuxLevel(	nMaxValOut	:= uiMaxLuxLevel,
					nValIn1		:= uiSPLuxLevel_MB,		//nValIn1 takes priotity in case of download or restart
					nValIn2		:= stRoomDataPLC.uiSpLuxLevel,
					nValOut		=> uiLuxOn
				);


fbWritePirDelayTIme(	nMaxValOut	:= uiMaxPirOffMinutes,
						nValIn1		:= uiPirOffDelayTime_MB,		//nValIn1 takes priotity in case of download or restart
						nValIn2		:= stRoomDataPLC.uiPirOffDelayTime,
						nValOut		=> uiPirOffMinutes
					);
					

//Convert read/write modbus data to appropriate datatypes in PLC
fLuxOn	:= TO_REAL(uiLuxOn);			
tPIROff	:= TO_TIME(uiPirOffMinutes*udTimeScaling); //Time conversion defaults to ms

fLuxDim	:= TO_REAL(stRoomDataPLC.uiSpDimLuxLevel);			
tPIRDim	:= TO_TIME(stRoomDataPLC.uiPirDimDelayTime*udTimeScaling); //Time conversion defaults to ms
END_ACTION

ACTION A_Sensor:

fbSensor.ipCommunication := P_DALI_Background.arrfbKL6821Communication[Sensor_DALI_LINE_NUM];

//only 1 sensor 
(*
fbSensor(
	byShrtAdr:= bySensorAddr,
	bInitialize:= bInitialize, 
	DALI_LINE_NUM:= Sensor_DALI_LINE_NUM, 
 	//bCancelHoldTimerOccupancy:= bCancelHoldTimerOccupancy, 
	stSensorSetup := stDaliSensorSetup,
	bInitErr=> bInitErr, 
	bInitDone=> bInitDone,
	stPirSensorData:= stPirSensorData, 
	arrSensorScales:= arrSensorScales);

*)
//several sensors	
fbSensor(
	arrShrtAdr:= arrSensorAddr,
	bInitialize:= bInitialize, 
	DALI_LINE_NUM:= Sensor_DALI_LINE_NUM, 
 	//bCancelHoldTimerOccupancy:= bCancelHoldTimerOccupancy, 
	stSensorSetup := stDaliSensorSetup,
	arrInitErr=> arrInitErr, 
	arrInitDone=> arrInitDone,
	stPirSensorData:= stPirSensorData, 
	arrSensorScales:= arrSensorScales);
END_ACTION

END_PROGRAM

// ---- POUs/Alle_Rum/Gange/Gang_5_441B/P_Gang_5_441B.TcPOU
PROGRAM P_Gang_5_441B
VAR

	arrfbLysGruppe			: ARRAY [1..2] OF FB_Light_Type_B;
	arrstDaliSetupGruppe	: ARRAY[1..2] OF SH_Light.ST_DALI_RoomSetup := 
	
													[(	byShrtAdr_Prim := 47, 
														byGrpAdr_Prim := 3, 
														eMod_Prim := E_DALIAddressType.Group, 
														//byShrtAdr_Sec := 1, 
														//byGrpAdr_Sec := 1, 
														//eMod_Sec := E_DALIAddressType.Short, 
														//byShrtAdr_Supl := 1,
														//eMod_Supl := E_DALIADDRESSTYPE.Group,
                                                        byGrpAdr_Supl := 1, 
														DALI_LINE_NUM_PRIM := arrDALI_LINE_NUM_LIGHT[1], 
														DALI_LINE_NUM_SEC := 0, //0 = ingen zonestyring/vinduerække
														DALI_LINE_NUM_SUPL := arrDALI_LINE_NUM_PENDANTS[1]),
														
													(	byShrtAdr_Prim := 1, 
														byGrpAdr_Prim := 3, 
														eMod_Prim := E_DALIAddressType.Group, 
														//byShrtAdr_Sec := 1, 
														//byGrpAdr_Sec := 1, 
														//eMod_Sec := E_DALIAddressType.Short, 
														//byShrtAdr_Supl := 1, 
														DALI_LINE_NUM_PRIM := arrDALI_LINE_NUM_LIGHT[2], 
														DALI_LINE_NUM_SEC := 0, 
														DALI_LINE_NUM_SUPL := arrDALI_LINE_NUM_PENDANTS[2])];
														
	arrstLiveDataGruppe		: ARRAY [1..2] OF SH_Light.ST_LiveData;
	//stLiveData AT %MB22	: SH_Light.ST_LiveData;
	
	arrRunTuningGruppe: ARRAY[1..2] OF BOOL;
	
	
	
	bTopButtonZone1			: BOOL;
	bTopButtonZone1_Visu	: BOOL;
	bBottomButtonZone1		: BOOL;
	bBottomButtonZone1_Visu	: BOOL;
	bButtonZone2			: BOOL;
	bNeighborRoomsPir		: BOOL;
	fLuxOn					: REAL; 
	fLuxDim					: REAL;
	tPIRDim					: TIME;
	tPIROff					: TIME;
	fOffsetSec				: REAL := 20;
    bOccupiedRoom		    : BOOL;;
//Digital In
//    bDigitalPir AT %I*      : BOOL ;    

// Sensor Settings
	//fbSensor					: SH_Light.FB_NIKO_P46xx_1Pcs;
	fbSensor					: SH_Light.FB_NIKO_P46xx_3Pcs;
	//bySensorAddr				: BYTE := 4;
	arrSensorAddr				: ARRAY[1..3] OF BYTE := [6,7,8];
	bInitialize					: BOOL := TRUE;
	stDaliSensorSetup			: ST_DALI_NIKOP46SetupData := (
																nSensitivityPIRSegmentA := arrSensitivityOccupancy[1],
																nSensitivityPIRSegmentB := arrSensitivityOccupancy[2],
																nSensitivityPIRSegmentC := arrSensitivityOccupancy[3]);
	//bInitErr					: BOOL;
	//bInitDone					: BOOL;
	arrInitErr					: ARRAY [1..3] OF BOOL;
	arrInitDone					: ARRAY [1..3] OF BOOL;
	arrSensorScales				: ARRAY [1..10] OF SH_Light.ST_DALI_SensorScaleMode := [	(fMeassureMaxSensor := 1023, fReadMaxSensor := 1023),
                                                                                            (fMeassureMaxSensor := 1023, fReadMaxSensor := 1023),
                                                                                            (fMeassureMaxSensor := 1023, fReadMaxSensor := 1023),																			
																						7(())];
	bCancelHoldTimerOccupancy	: BOOL;
(*	eEventPriorityOccupancy		: E_DALIEventPriority := E_DALIEVENTPRIORITY.Middle;
	nHoldTimerOccupancy			: WORD := 5; // Value in s. 	
	nReportTimerOccupancy		: BYTE := 120; // Value in s, Preset manufacturer value
	nDeadtimeTimerOccupancy		: WORD := 100; // Value in ms, Predefined Value of DALI Standard
	bCancelHoldTimerOccupancy	: BOOL;
	nSensitivityOccupancy		: BYTE:= 3; //setting Sensivity (0..4) 0 (Off), 1 (Min), 2(Low), 3(High) and 4 (Max)

	bEnableLuxEvent				: BOOL;
	eEventPriorityBrightness	: E_DALIEventPriority := E_DALIEVENTPRIORITY.Middle;
	nDeadtimeTimerBrightness	: WORD := 1500; // Value in ms, Predefined Value of DALI Standard
	nHysteresisBrightness		: BYTE := 2; // Value in %
	nHysteresisMinBrightness	: BYTE := 10; // Absolute Value, depending on the manufacturer specific resolution
	nReportTimerBrightness		: BYTE := 120; // Value in s, Preset manufacturer value
*)


//ModbusComm setup
	
	fbWriteSPLuxLevel			: SH_Light.FB_TwoVal_SelectOne_RTrigChange;
	fbWritePirDelayTIme			: SH_Light.FB_TwoVal_SelectOne_RTrigChange;
	stRoomDataPLC				: SH_Light.ST_RoomDataPLC	:=	(	uiPirOffDelayTime	:= 30,
																	uiSpLuxLevel		:= 500,
																	uiPirDimDelayTime	:= 15,
																	uiSpDimLuxLevel		:= 200
																);
	fbBallastOnHours			: SH_Light.FB_CountOnHours;
	bEnableHourCount			: BOOL := TRUE;
	
	//Non-persistent modbus data
	bPirActive_MB			AT%MX196.0	: BOOL;				//bPirLys i gammel kode
	uiActLuxLevel_MB		AT%MB200	: UINT;				//intHMIAktueltLux i gammel kode
	uiActLightLevelPct_MB	AT%MB206	: UINT;				//intDALI_Gruppe1_Lysniveau i gammel kode
	
	//For Conversion
	uiPirOffMinutes						: UINT;
	udTimeScaling						: UDINT := 60000;
	uiLuxOn								: UINT;
	
	//max values checks
	uiMaxLuxLevel						: UINT := 1023;
	uiMaxPirOffMinutes					: UINT := 180;
	
END_VAR

VAR CONSTANT
	Sensor_DALI_LINE_NUM: BYTE := 3;
	arrDALI_LINE_NUM_LIGHT: ARRAY[1..2] OF BYTE := [1,2]; //korrekt rækkefølge nødvendig //rækkefølge og linje 
	arrDALI_LINE_NUM_PENDANTS: ARRAY[1..2] OF BYTE := [0,0]; //korrekt rækkefølge nødvendig. 0 = ingen pendler
	arrSensitivityOccupancy				: ARRAY[1..3] OF BYTE := [4,4,4];
END_VAR
VAR PERSISTENT
	stPirSensorData: SH_Light.ST_DALI_Sensor;
	arrstTuneDataGruppe: ARRAY [1..2] OF SH_Light.ST_TuneData_EX;

	uiPirOffDelayTime_MB	AT%MB198	    : UINT;				//intHMI_Pir_SetValue i gammel kode
	uiSPLuxLevel_MB		    AT%MB202     : UINT;				//intHMI_Lux_SetValue i gammel kode
	uiBallastOnHours_MB	    AT%MB210	    : UINT;				//dintHMILysbraendtimer1 i gammel kode
	byOnHoursOverflowCount			    : BYTE;
END_VAR

///////)

A_Buttons();
A_LightCtrl();
A_ModbusComm();
A_Sensor();

ACTION A_Buttons:
bTopButtonZone1		:= GVL_EnOcean.strEnOceanSwitch_Gang_5_441B.bT2_ON OR bTopButtonZone1_Visu;
bBottomButtonZone1	:= GVL_EnOcean.strEnOceanSwitch_Gang_5_441B.bT2_OFF OR bBottomButtonZone1_Visu;
END_ACTION

ACTION A_LightCtrl:
bNeighborRoomsPir	:= P_Rum_5_441A.stPirSensorData.bPrc              OR
                       P_Rum_5_448b.stPirSensorData.bPrc              OR
					   P_Rum_5_444.stPirSensorData.bPrc               OR
					   P_Gang_4_413.stPirSensorData.bPrc               ;
					   
					   
					   
					   
//gruppe 6
arrfbLysGruppe[1]( 
	nZoneID:= 1, 
	bButtonZone1:= bTopButtonZone1,
	bBottomButtonZone1 := bBottomButtonZone1,
	//bButtonZone2:= bButtonZone2,
	//bNoButtons := TRUE,
	bNeighborRoomsPir	:=	bNeighborRoomsPir,
	fLuxOn:= fLuxOn, 
	fLuxDim:= fLuxDim, 
	tPIRDim:= tPIRDim, 
	tPIROff:= tPIROff, 
	fOffsetSec:= fOffsetSec, 
	bReInit:= , 
	stDaliSetup:= arrstDaliSetupGruppe[1], 
	ipCommunication_Prim:= P_DALI_Background.arrfbKL6821Communication[arrDALI_LINE_NUM_LIGHT[1]], 
	//ipCommunication_Sec:= P_DALI_Background.arrfbKL6821Communication[arrDALI_LINE_NUM_LIGHT[1]], //samme som lyslinjen, hvis den ikke eksisterer
	//ipCommunication_Supl:= P_DALI_Background.arrfbKL6821Communication[arrDALI_LINE_NUM_LIGHT[1]],//samme som lyslinjen, hvis den ikke eksisterer 
	fMinOutputPowerLevelRoom:= 15, 
	fMaxOutputPowerLevelRoom:= 100, 
	nCycleTimeInMS:= SH_Light.DALI_Param.nPlcTaskCycleTimeInMS*nDimCmdCycleTimeFactor,  //Used only for dim. Factor=2 makes dimming smooth
	bRunTuning:= arrRunTuningGruppe[1], 
	bOccupiedRoom=> , 
	bError_Prim=> , 
	nError_Prim=> , 
	stTuneData:=arrstTuneDataGruppe[1] , 
	stPirSensorData:= stPirSensorData, 					//samme sensordata
	stLiveData:= arrstLiveDataGruppe[1]);

//gruppe 15	
arrfbLysGruppe[2]( 
	nZoneID:= 1, 
	bButtonZone1:= bTopButtonZone1,
	bBottomButtonZone1 := bBottomButtonZone1,
	//bButtonZone2:= bButtonZone2,
	//bNoButtons := TRUE,
	bNeighborRoomsPir	:=	bNeighborRoomsPir,
	fLuxOn:= fLuxOn, 
	fLuxDim:= fLuxDim, 
	tPIRDim:= tPIRDim, 
	tPIROff:= tPIROff, 
	fOffsetSec:= fOffsetSec, 
	bReInit:= , 
	stDaliSetup:= arrstDaliSetupGruppe[2], 
	ipCommunication_Prim:= P_DALI_Background.arrfbKL6821Communication[arrDALI_LINE_NUM_LIGHT[2]], 
	//ipCommunication_Sec:= P_DALI_Background.arrfbKL6821Communication[arrDALI_LINE_NUM_LIGHT[2]], //samme som lyslinjen, hvis den ikke eksisterer
	//ipCommunication_Supl:= P_DALI_Background.arrfbKL6821Communication[arrDALI_LINE_NUM_LIGHT[2]], //samme som lyslinjen, hvis den ikke eksisterer 
	fMinOutputPowerLevelRoom:= 15, 
	fMaxOutputPowerLevelRoom:= 100, 
	nCycleTimeInMS:= SH_Light.DALI_Param.nPlcTaskCycleTimeInMS*nDimCmdCycleTimeFactor,  //Used only for dim. Factor=2 makes dimming smooth
	bRunTuning:= arrRunTuningGruppe[2], 
	bOccupiedRoom=> , 
	bError_Prim=> , 
	nError_Prim=> , 
	stTuneData:=arrstTuneDataGruppe[2] , 
	stPirSensorData:= stPirSensorData, 					//samme sensordata
	stLiveData:= arrstLiveDataGruppe[2]);
END_ACTION

ACTION A_ModbusComm:
//Manage data for modbus communication

//Manage data for read-only in PLC
stRoomDataPLC.bPirActive			:= stPirSensorData.bPrc;
stRoomDataPLC.uiActLuxLevel			:= TO_UINT(TRUNC(stPirSensorData.fBrightness));
stRoomDataPLC.uiActLightLevelPct	:= TO_UINT(TRUNC(arrfbLysGruppe[1].fbBallast.fActlLgtLvl_Prim));
		//stRoomDataPLC.uiActLightLevelPct	:= TO_UINT(TRUNC(fbLys.fbBallast.fActlLgtLvl_Prim)); //if only one group light control
stRoomDataPLC.uiBallastOnHours		:= uiBallastOnHours_MB; //The calculation for BallastOnHours is stored directly to the MB register below


//Assign data for read-only to MB registers
bPirActive_MB		:= stRoomDataPLC.bPirActive;
uiActLuxLevel_MB	:= stRoomDataPLC.uiActLuxLevel;

	//calculate BallastOnHours
	fbBallastOnHours(
		bEnableHourCount	:= bEnableHourCount,
		bPauseCount			:= arrfbLysGruppe[1].fbLightCtrl.bOffZone1,
		uiOnHours			:= uiBallastOnHours_MB,			//OnHours is updated here
		byOverflowCount		:= byOnHoursOverflowCount);


//Manage data for read/write for both PLC and MB registers
fbWriteSPLuxLevel(	nMaxValOut	:= uiMaxLuxLevel,
					nValIn1		:= uiSPLuxLevel_MB,		//nValIn1 takes priotity in case of download or restart
					nValIn2		:= stRoomDataPLC.uiSpLuxLevel,
					nValOut		=> uiLuxOn
				);


fbWritePirDelayTIme(	nMaxValOut	:= uiMaxPirOffMinutes,
						nValIn1		:= uiPirOffDelayTime_MB,		//nValIn1 takes priotity in case of download or restart
						nValIn2		:= stRoomDataPLC.uiPirOffDelayTime,
						nValOut		=> uiPirOffMinutes
					);
					

//Convert read/write modbus data to appropriate datatypes in PLC
fLuxOn	:= TO_REAL(uiLuxOn);			
tPIROff	:= TO_TIME(uiPirOffMinutes*udTimeScaling); //Time conversion defaults to ms

fLuxDim	:= TO_REAL(stRoomDataPLC.uiSpDimLuxLevel);			
tPIRDim	:= TO_TIME(stRoomDataPLC.uiPirDimDelayTime*udTimeScaling); //Time conversion defaults to ms
END_ACTION

ACTION A_Sensor:

fbSensor.ipCommunication := P_DALI_Background.arrfbKL6821Communication[Sensor_DALI_LINE_NUM];
(*
//only 1 sensor
fbSensor(
	byShrtAdr:= bySensorAddr,
	bInitialize:= bInitialize, 
	DALI_LINE_NUM:= Sensor_DALI_LINE_NUM, 
 	//bCancelHoldTimerOccupancy:= bCancelHoldTimerOccupancy, 
	stSensorSetup := stDaliSensorSetup,
	bInitErr=> bInitErr, 
	bInitDone=> bInitDone,
	stPirSensorData:= stPirSensorData, 
	arrSensorScales:= arrSensorScales);
	*)

//several sensors	
fbSensor(
	arrShrtAdr:= arrSensorAddr,
	bInitialize:= bInitialize, 
	DALI_LINE_NUM:= Sensor_DALI_LINE_NUM, 
 	//bCancelHoldTimerOccupancy:= bCancelHoldTimerOccupancy, 
	stSensorSetup := stDaliSensorSetup,
	arrInitErr=> arrInitErr, 
	arrInitDone=> arrInitDone,
	stPirSensorData:= stPirSensorData, 
	arrSensorScales:= arrSensorScales);
END_ACTION

END_PROGRAM

// ---- POUs/Alle_Rum/Rum_Med_DALI_Pir/1Rum_5_448B/P_Rum_5_448B.TcPOU
PROGRAM P_Rum_5_448B
VAR

	fbLys		: FB_Light_Type_B;
	
	stDaliSetup	: SH_Light.ST_DALI_RoomSetup := (
														byShrtAdr_Prim := 21, 
														byGrpAdr_Prim := 5, 
														eMod_Prim := E_DALIAddressType.Group, 
														//byShrtAdr_Sec := 1, 
														//byGrpAdr_Sec := 1, 
														//eMod_Sec := E_DALIAddressType.Short, 
														//byShrtAdr_Supl := 1,
														//byGrpAdr_Supl := 1,
														//eMod_Prim := E_DALIAddressType.Short 
														DALI_LINE_NUM_PRIM := DALI_LINE_NUM_LIGHT, 
														DALI_LINE_NUM_SEC := 0, //0 = ingen zonestyring/vinduerække
														DALI_LINE_NUM_SUPL := DALI_LINE_NUM_PENDANTS);
														
	stLiveData				: SH_Light.ST_LiveData;
	bRunTuning					: BOOL;
	
	bTopButtonZone1				: BOOL;
	bTopButtonZone1_Visu		: BOOL;
	bBottomButtonZone1			: BOOL;
	bBottomButtonZone1_Visu	    : BOOL;
	bButtonZone2				: BOOL;
	bNeighborRoomsPir		    : BOOL;
	fLuxOn				     	: REAL;
	fLuxDim						: REAL;
	tPIRDim						: TIME;
	tPIROff						: TIME;
	fOffsetSec					: REAL := 20;
	bOccupiedRoom			    : BOOL;


// Sensor Settings
	fbSensor						: SH_Light.FB_NIKO_P46xx_1Pcs;
	//fbSensor						: SH_Light.FB_NIKO_P46xx_3Pcs;
	bySensorAddr				    : BYTE := 8;
	//arrSensorAddr				    : ARRAY[1..3] OF BYTE := [7,8,9];
	bInitialize						: BOOL := TRUE;
	stDaliSensorSetup			    : ST_DALI_NIKOP46SetupData := (
																nSensitivityPIRSegmentA := arrSensitivityOccupancy[1],
																nSensitivityPIRSegmentB := arrSensitivityOccupancy[2],
																nSensitivityPIRSegmentC := arrSensitivityOccupancy[3]);
	bInitErr						: BOOL;
	bInitDone						: BOOL;
	//arrInitErr					: ARRAY [1..3] OF BOOL;
	//arrInitDone					: ARRAY [1..3] OF BOOL;
	arrSensorScales				    : ARRAY [1..10] OF SH_Light.ST_DALI_SensorScaleMode := [
																						(fMeassureMaxSensor := 1023, fReadMaxSensor := 1023),																																										
																						9(())];
	bCancelHoldTimerOccupancy	: BOOL;
(*	eEventPriorityOccupancy		: E_DALIEventPriority := E_DALIEVENTPRIORITY.Middle;
	nHoldTimerOccupancy			: WORD := 5; // Value in s. 	
	nReportTimerOccupancy		: BYTE := 120; // Value in s, Preset manufacturer value
	nDeadtimeTimerOccupancy		: WORD := 100; // Value in ms, Predefined Value of DALI Standard
	bCancelHoldTimerOccupancy	: BOOL;
	nSensitivityOccupancy		: BYTE:= 3; //setting Sensivity (0..4) 0 (Off), 1 (Min), 2(Low), 3(High) and 4 (Max)

	bEnableLuxEvent				: BOOL;
	eEventPriorityBrightness	: E_DALIEventPriority := E_DALIEVENTPRIORITY.Middle;
	nDeadtimeTimerBrightness	: WORD := 1500; // Value in ms, Predefined Value of DALI Standard
	nHysteresisBrightness		: BYTE := 2; // Value in %
	nHysteresisMinBrightness	: BYTE := 10; // Absolute Value, depending on the manufacturer specific resolution
	nReportTimerBrightness		: BYTE := 120; // Value in s, Preset manufacturer value
*)

	//stDaliSetup: SH_Light.ST_DALI_RoomSetup
	//stRoomDataModbus			: SH_Light.ST_RoomDataModbus := ( bPirActive := bPirActive
	

	//ModbusComm setup
	
	fbWriteSPLuxLevel			: SH_Light.FB_TwoVal_SelectOne_RTrigChange;
	fbWritePirDelayTIme		: SH_Light.FB_TwoVal_SelectOne_RTrigChange;
	stRoomDataPLC				: SH_Light.ST_RoomDataPLC	:=	(
																	uiPirOffDelayTime	:= 30,
																	uiSpLuxLevel			:= 500,
																	uiPirDimDelayTime	:= 15,
																	uiSpDimLuxLevel		:= 200);
																	
	fbBallastOnHours				: SH_Light.FB_CountOnHours;
	bEnableHourCount			: BOOL := TRUE;
	
	//Non-persistent modbus data
	bPirActive_MB				AT %MX94.0	: BOOL;				//bPirLys i gammel kode
	uiActLuxLevel_MB			AT %MB548	: UINT;				//intHMIAktueltLux i gammel kode
	uiActLightLevelPct_MB	    AT %MB98	: UINT;				//intDALI_Gruppe1_Lysniveau i gammel kode
	
	//For Conversion
	uiPirOffMinutes						: UINT;
	udTimeScaling						: UDINT := 60000;
	uiLuxOn								: UINT;
	
	//max values checks
	uiMaxLuxLevel						: UINT := 1023;
	uiMaxPirOffMinutes				: UINT := 180;

	
END_VAR

VAR CONSTANT
    Sensor_DALI_LINE_NUM				: BYTE := 4;
	DALI_LINE_NUM_LIGHT			     	: BYTE := 2;
	DALI_LINE_NUM_PENDANTS	            : BYTE := 0; //0=ingen pendler	
	arrSensitivityOccupancy				: ARRAY[1..3] OF BYTE := [4,4,4];
END_VAR
VAR PERSISTENT
	stPirSensorData: SH_Light.ST_DALI_Sensor;
	stTuneData: SH_Light.ST_TuneData_EX;

	uiPirOffDelayTime_MB	AT %MB96	: UINT;				//ntHMI_Pir_SetValue i gammel kode
	uiSPLuxLevel_MB			AT %MB550	: UINT;				//intHMI_Lux_SetValue i gammel kode
	uiBallastOnHours_MB		AT %MB100	: UINT;				//dintHMILysbraendtimer1 i gammel kode
	byOnHoursOverflowCount				: BYTE;   
END_VAR

A_Buttons();
A_LightCtrl();
A_Sensor();
A_ModbusComm();

ACTION A_Buttons:
bTopButtonZone1		:= GVL_EnOcean.strEnOceanSwitch_Rum_5_448A.bT2_ON OR bTopButtonZone1_Visu;
bBottomButtonZone1	:= GVL_EnOcean.strEnOceanSwitch_Rum_5_448A.bT2_OFF OR bBottomButtonZone1_Visu;
END_ACTION

ACTION A_LightCtrl:

